Omron Sysmac Studio project TestDataGenerator (Sysmac Studio 1.66.0.7, StandardProject)

# Controller Util: NX102-9000 version 1.64
Task PrimaryTask (priority 4, period or condition 10000): Generate
Library RingBufferLib 0.0.2 (contents left out)
Library FileStreamWriterLib 0.0.2 (contents left out)

TYPE Alignment1Struct : STRUCT  (* Size = 4; Tail Padding = 0; Alignment = 1; Density = 1.000; *)
    aUsint : USINT;  (* Offset = 0; Padding = 0; Size = 1; Alignment = 1; *)
    aSint : SINT;  (* Offset = 1; Padding = 0; Size = 1; Alignment = 1; *)
    Bytes : ARRAY[0..1] OF BYTE;  (* Offset = 2; Padding = 0; Size = 2; Alignment = 1; *)
END_STRUCT END_TYPE
TYPE Alignment2Struct : STRUCT  (* Size = 8; Tail Padding = 0; Alignment = 2; Density = 0.578; *)
    aBool : BOOL;  (* Offset = 0; Padding = 0; Size = 2; Alignment = 2; *)
    aUint : UINT;  (* Offset = 2; Padding = 0; Size = 2; Alignment = 2; *)
    aInt : INT;  (* Offset = 4; Padding = 0; Size = 2; Alignment = 2; *)
    Bools : ARRAY[0..3] OF BOOL;  (* Offset = 6; Padding = 0; Size = 2; Alignment = 2; *)
END_STRUCT END_TYPE
TYPE Alignment4Struct : STRUCT  (* Size = 16; Tail Padding = 0; Alignment = 4; Density = 1.000; *)
    aUdint : UDINT;  (* Offset = 0; Padding = 0; Size = 4; Alignment = 4; *)
    aDint : DINT;  (* Offset = 4; Padding = 0; Size = 4; Alignment = 4; *)
    Uints : ARRAY[0..1] OF UINT;  (* Offset = 8; Padding = 0; Size = 4; Alignment = 2; *)
    Bytes : ARRAY[0..3] OF BYTE;  (* Offset = 12; Padding = 0; Size = 4; Alignment = 1; *)
END_STRUCT END_TYPE
TYPE Alignment8Struct : STRUCT  (* Size = 32; Tail Padding = 0; Alignment = 8; Density = 0.895; *)
    aUlint : ULINT;  (* Offset = 0; Padding = 0; Size = 8; Alignment = 8; *)
    aLint : LINT;  (* Offset = 8; Padding = 0; Size = 8; Alignment = 8; *)
    Udints : ARRAY[0..1] OF UDINT;  (* Offset = 16; Padding = 0; Size = 8; Alignment = 4; *)
    aAlignment2Struct : Alignment2Struct;  (* Offset = 24; Padding = 0; Size = 8; Alignment = 2; *)
END_STRUCT END_TYPE
TYPE SmallStruct : STRUCT  (* Size = 6; Tail Padding = 0; Alignment = 1; Density = 0.857 *)
    u : USINT;  (* Offset = 0; Padding = 0; Size = 1; Alignment = 1; *)
    s : STRING[5];  (* Offset = 1; Padding = 0; Size = 5; Alignment = 1; *)
END_STRUCT END_TYPE
TYPE PaddedStruct : STRUCT  (* Size = 32; Tail Padding = 6; Alignment = 8; Density = 0.466; *)
    aUsint : USINT;  (* Offset = 0; Padding = 0; Size = 1; Alignment = 1; *)
    aUint : UINT;  (* Offset = 2; Padding = 1; Size = 2; Alignment = 2; *)
    aSint : SINT;  (* Offset = 5; Padding = 0; Size = 1; Alignment = 1; *)
    aDint : DINT;  (* Offset = 8; Padding = 2; Size = 4; Alignment = 4; *)
    aUlint : ULINT;  (* Offset = 16; Padding = 4; Size = 8; Alignment = 8; *)
    aBool : BOOL;  (* Offset = 24; Padding = 0; Size = 2; Alignment = 2; *)
END_STRUCT END_TYPE
TYPE UnionStruct : STRUCT  (* Size = 32; Tail Padding = 0; Alignment = 8; Density = 1.000; *)
    Alignment1Unions : ARRAY[0..1] OF Alignment1Union;  (* Offset = 0; Padding = 0; Size = 8; Alignment = 1; *)
    Alignment2Unions : ARRAY[0..1] OF Alignment2Union;  (* Offset = 8; Padding = 0; Size = 8; Alignment = 2; *)
    aAlignment4Union : Alignment4Union;  (* Offset = 16; Padding = 0; Size = 8; Alignment = 4; *)
    aAlignment8Union : Alignment8Union;  (* Offset = 24; Padding = 0; Size = 8; Alignment = 8; *)
END_STRUCT END_TYPE
TYPE ComplexStruct : STRUCT  (* Size = 56; Tail Padding = 4; Alignment = 8; Density = 0.806; *)
    aUsint : USINT;  (* Offset = 0; Padding = 0; Size = 1; Alignment = 1; *)
    Alignment2Structs : ARRAY[0..1] OF Alignment2Struct;  (* Offset = 2; Padding = 1; Size = 16; Alignment = 2; *)
    aAlignment4Union : Alignment4Union;  (* Offset = 20; Padding = 2; Size = 8; Alignment = 4; *)
    aBool : BOOL;  (* Offset = 28; Padding = 0; Size = 2; Alignment = 2; *)
    Lints : ARRAY[0..1] OF LINT;  (* Offset = 32; Padding = 2; Size = 16; Alignment = 8; *)
    aEnum : TestEnum;  (* Offset = 52; Padding = 0; Size = 4; Alignment = 4; *)
END_STRUCT END_TYPE
TYPE Nest1Struct : STRUCT  (* Size = 8; Tail Padding = 0; Alignment = 2; Density = 1.000; *)
    aSmallStruct : SmallStruct;  (* Offset = 0; Padding = 0; Size = 6; Alignment = 1; *)
    aInt : INT;  (* Offset = 6; Padding = 0; Size = 2; Alignment = 2; *)
END_STRUCT END_TYPE
TYPE Nest2Struct : STRUCT  (* Size = 20; Tail Padding = 0; Alignment = 4; Density =0.900; *)
    aNest1Struct : Nest1Struct;  (* Offset = 0; Padding = 0; Size = 8; Alignment = 2; *)
    aSmallStruct : SmallStruct;  (* Offset = 8; Padding = 0; Size = 6; Alignment = 1; *)
    aDint : DINT;  (* Offset = 16; Padding = 2; Size = 4; Alignment = 4; *)
END_STRUCT END_TYPE
TYPE Nest3Struct : STRUCT  (* Size = 40; Tail Padding = 0; Alignment = 8; Density =0.800; *)
    aNest2Struct : Nest2Struct;  (* Offset = 0; Padding = 0; Size = 20; Alignment = 4; *)
    aSmallStruct : SmallStruct;  (* Offset = 20; Padding = 0; Size = 6; Alignment = 1; *)
    aLint : LINT;  (* Offset = 32; Padding = 6; Size = 8; Alignment = 8; *)
END_STRUCT END_TYPE
TYPE ExampleStruct : STRUCT  (* Size = 32; Tail Padding = 4; Alignment = 8; Density =0.875; *)
    Vel : LREAL;  (* Offset = 0; Padding = 0; Size = 8; Alignment = 8; *)
    Trq : LREAL;  (* Offset = 8; Padding = 0; Size = 8; Alignment = 8; *)
    Acc : LREAL;  (* Offset = 16; Padding = 0; Size = 8; Alignment = 8; *)
    StatusCode : DWORD;  (* Offset = 24; Padding = 0; Size = 4; Alignment = 4; *)
END_STRUCT END_TYPE
TYPE Alignment1Union1D : STRUCT
    Unions : ARRAY[0..2] OF Alignment1Union;
END_STRUCT END_TYPE
TYPE Alignment1Union2D : STRUCT
    Unions : ARRAY[0..2,0..2] OF Alignment1Union;
END_STRUCT END_TYPE
TYPE Alignment1Union3D : STRUCT
    Unions : ARRAY[0..2,0..2,0..2] OF Alignment1Union;
END_STRUCT END_TYPE
TYPE Alignment1UnionD1E1 : STRUCT
    Unions : ARRAY[0..0] OF Alignment1Union;
END_STRUCT END_TYPE
TYPE Alignment1UnionD2E1 : STRUCT
    Unions : ARRAY[0..0,0..0] OF Alignment1Union;
END_STRUCT END_TYPE
TYPE Alignment1UnionD3E1 : STRUCT
    Unions : ARRAY[0..0,0..0,0..0] OF Alignment1Union;
END_STRUCT END_TYPE
TYPE Alignment2Union1D : STRUCT
    Unions : ARRAY[0..2] OF Alignment2Union;
END_STRUCT END_TYPE
TYPE Alignment2Union2D : STRUCT
    Unions : ARRAY[0..2,0..2] OF Alignment2Union;
END_STRUCT END_TYPE
TYPE Alignment2Union3D : STRUCT
    Unions : ARRAY[0..2,0..2,0..2] OF Alignment2Union;
END_STRUCT END_TYPE
TYPE Alignment2UnionD1E1 : STRUCT
    Unions : ARRAY[0..0] OF Alignment2Union;
END_STRUCT END_TYPE
TYPE Alignment2UnionD2E1 : STRUCT
    Unions : ARRAY[0..0,0..0] OF Alignment2Union;
END_STRUCT END_TYPE
TYPE Alignment2UnionD3E1 : STRUCT
    Unions : ARRAY[0..0,0..0,0..0] OF Alignment2Union;
END_STRUCT END_TYPE
TYPE Alignment4Union1D : STRUCT
    Unions : ARRAY[0..2] OF Alignment4Union;
END_STRUCT END_TYPE
TYPE Alignment1Union : UNION  (* Size = 4; Padding = 0; Alignment = 1; Density = 1.000 *)
    Bytes : ARRAY[0..3] OF BYTE;  (* Offset = 0; Padding = 0; Size = 4; Alignment = 1; *)
END_UNION END_TYPE
TYPE Alignment2Union : UNION  (* Size = 4; Padding = 0; Alignment = 2; Density = 1.000 *)
    aBool : BOOL;  (* Offset = 0; Padding = 0; Size = 2; Alignment = 2; *)
    Words : ARRAY[0..1] OF WORD;  (* Offset = 0; Padding = 0; Size = 4; Alignment = 2; *)
END_UNION END_TYPE
TYPE Alignment4Union : UNION  (* Size = 8; Padding = 0; Alignment = 4; Density = 1.000 *)
    Bytes : ARRAY[0..3] OF BYTE;  (* Offset = 0; Padding = 0; Size = 4; Alignment = 1; *)
    Dwords : ARRAY[0..1] OF DWORD;  (* Offset = 0; Padding = 0; Size = 8; Alignment = 4; *)
END_UNION END_TYPE
TYPE Alignment8Union : UNION  (* Size = 8; Padding = 0; Alignment = 8; Density = 1.000 *)
    Words : ARRAY[0..3] OF WORD;  (* Offset = 0; Padding = 0; Size = 8; Alignment = 2; *)
    aLword : LWORD;  (* Offset = 0; Padding = 0; Size = 8; Alignment = 8; *)
END_UNION END_TYPE
TYPE MyEnum : (E1 := 0, E2 := 1); END_TYPE
TYPE MyEnum2 : (E2_1 := 0, E2_2 := 1); END_TYPE
TYPE Alignment4Union2D : STRUCT
    Unions : ARRAY[0..2,0..2] OF Alignment4Union;
END_STRUCT END_TYPE
TYPE Alignment4Union3D : STRUCT
    Unions : ARRAY[0..2,0..2,0..2] OF Alignment4Union;
END_STRUCT END_TYPE
TYPE Alignment4UnionD1E1 : STRUCT
    Unions : ARRAY[0..0] OF Alignment4Union;
END_STRUCT END_TYPE
TYPE Alignment4UnionD2E1 : STRUCT
    Unions : ARRAY[0..0,0..0] OF Alignment4Union;
END_STRUCT END_TYPE
TYPE Alignment4UnionD3E1 : STRUCT
    Unions : ARRAY[0..0,0..0,0..0] OF Alignment4Union;
END_STRUCT END_TYPE
TYPE Alignment8Union1D : STRUCT
    Unions : ARRAY[0..2] OF Alignment8Union;
END_STRUCT END_TYPE
TYPE Alignment8Union2D : STRUCT
    Unions : ARRAY[0..2,0..2] OF Alignment8Union;
END_STRUCT END_TYPE
TYPE Alignment8Union3D : STRUCT
    Unions : ARRAY[0..2,0..2,0..2] OF Alignment8Union;
END_STRUCT END_TYPE
TYPE Alignment8UnionD1E1 : STRUCT
    Unions : ARRAY[0..0] OF Alignment8Union;
END_STRUCT END_TYPE
TYPE Alignment8UnionD2E1 : STRUCT
    Unions : ARRAY[0..0,0..0] OF Alignment8Union;
END_STRUCT END_TYPE
TYPE Alignment8UnionD3E1 : STRUCT
    Unions : ARRAY[0..0,0..0,0..0] OF Alignment8Union;
END_STRUCT END_TYPE
TYPE TestEnum : (TE_E0 := 0, TE_E1 := 1); END_TYPE
TYPE ExampleUnion : UNION  (* Size = 4; Padding = 0; Alignment = 4; Density = 1.000 *)
    StatusFlags : ARRAY[0..15] OF BOOL;  (* Offset = 0; Padding = 0; Size = 2; Alignment = 2; *)
    SegmentedStatusCodes : ARRAY[0..1] OF WORD;  (* Offset = 0; Padding = 0; Size = 4; Alignment = 2; *)
    StatusCode : DWORD;  (* Offset = 0; Padding = 0; Size = 4; Alignment = 4; *)
END_UNION END_TYPE

PROGRAM Generate
VAR
    iFileWriteVar : FileWriteVar;
    iFileWriter : stfreakjp\fileio\FileStreamWriter;
END_VAR
VAR CONSTANT
    STATE_INIT : UINT := 0;
    STATE_CREATE_TEST_VAR : UINT := 20;
    STATE_FINALIZE : UINT := 900;
    STATE_DONE : UINT := 1000;
END_VAR
VAR
    WRITE_VAR_BASE_PATH : STRING[65];
    VARS_LIST_PS1 : STRING[65];
    USINT_ARR_D1 : ARRAY[0..2] OF USINT;
    USINT_ARR_D2 : ARRAY[0..2,0..2] OF USINT;
    USINT_ARR_D3 : ARRAY[0..2,0..2,0..2] OF USINT;
    USINT_ARR_D1_E1 : ARRAY[0..0] OF USINT;
    USINT_ARR_D2_E1 : ARRAY[0..0,0..0] OF USINT;
    USINT_ARR_D3_E1 : ARRAY[0..0,0..0,0..0] OF USINT;
    UINT_ARR_D1 : ARRAY[0..2] OF UINT;
    UINT_ARR_D2 : ARRAY[0..2,0..2] OF UINT;
    UINT_ARR_D3 : ARRAY[0..2,0..2,0..2] OF UINT;
    UINT_ARR_D1_E1 : ARRAY[0..0] OF UINT;
    UINT_ARR_D2_E1 : ARRAY[0..0,0..0] OF UINT;
    UINT_ARR_D3_E1 : ARRAY[0..0,0..0,0..0] OF UINT;
    UDINT_ARR_D1 : ARRAY[0..2] OF UDINT;
    UDINT_ARR_D2 : ARRAY[0..2,0..2] OF UDINT;
    UDINT_ARR_D3 : ARRAY[0..2,0..2,0..2] OF UDINT;
    UDINT_ARR_D1_E1 : ARRAY[0..0] OF UDINT;
    UDINT_ARR_D2_E1 : ARRAY[0..0,0..0] OF UDINT;
    UDINT_ARR_D3_E1 : ARRAY[0..0,0..0,0..0] OF UDINT;
    ULINT_ARR_D1 : ARRAY[0..2] OF ULINT;
    ULINT_ARR_D2 : ARRAY[0..2,0..2] OF ULINT;
    ULINT_ARR_D3 : ARRAY[0..2,0..2,0..2] OF ULINT;
    ULINT_ARR_D1_E1 : ARRAY[0..0] OF ULINT;
    ULINT_ARR_D2_E1 : ARRAY[0..0,0..0] OF ULINT;
    ULINT_ARR_D3_E1 : ARRAY[0..0,0..0,0..0] OF ULINT;
    SINT_ARR_D1 : ARRAY[0..2] OF SINT;
    SINT_ARR_D2 : ARRAY[0..2,0..2] OF SINT;
    SINT_ARR_D3 : ARRAY[0..2,0..2,0..2] OF SINT;
    SINT_ARR_D1_E1 : ARRAY[0..0] OF SINT;
    SINT_ARR_D2_E1 : ARRAY[0..0,0..0] OF SINT;
    SINT_ARR_D3_E1 : ARRAY[0..0,0..0,0..0] OF SINT;
    INT_ARR_D1 : ARRAY[0..2] OF INT;
    INT_ARR_D2 : ARRAY[0..2,0..2] OF INT;
    INT_ARR_D3 : ARRAY[0..2,0..2,0..2] OF INT;
    INT_ARR_D1_E1 : ARRAY[0..0] OF INT;
    INT_ARR_D2_E1 : ARRAY[0..0,0..0] OF INT;
    INT_ARR_D3_E1 : ARRAY[0..0,0..0,0..0] OF INT;
    DINT_ARR_D1 : ARRAY[0..2] OF DINT;
    DINT_ARR_D2 : ARRAY[0..2,0..2] OF DINT;
    DINT_ARR_D3 : ARRAY[0..2,0..2,0..2] OF DINT;
    DINT_ARR_D1_E1 : ARRAY[0..0] OF DINT;
    DINT_ARR_D2_E1 : ARRAY[0..0,0..0] OF DINT;
    DINT_ARR_D3_E1 : ARRAY[0..0,0..0,0..0] OF DINT;
    LINT_ARR_D1 : ARRAY[0..2] OF LINT;
    LINT_ARR_D2 : ARRAY[0..2,0..2] OF LINT;
    LINT_ARR_D3 : ARRAY[0..2,0..2,0..2] OF LINT;
    LINT_ARR_D1_E1 : ARRAY[0..0] OF LINT;
    LINT_ARR_D2_E1 : ARRAY[0..0,0..0] OF LINT;
    LINT_ARR_D3_E1 : ARRAY[0..0,0..0,0..0] OF LINT;
    BYTE_ARR_D1 : ARRAY[0..2] OF BYTE;
    BYTE_ARR_D2 : ARRAY[0..2,0..2] OF BYTE;
    BYTE_ARR_D3 : ARRAY[0..2,0..2,0..2] OF BYTE;
    BYTE_ARR_D1_E1 : ARRAY[0..0] OF BYTE;
    BYTE_ARR_D2_E1 : ARRAY[0..0,0..0] OF BYTE;
    BYTE_ARR_D3_E1 : ARRAY[0..0,0..0,0..0] OF BYTE;
    WORD_ARR_D1 : ARRAY[0..2] OF WORD;
    WORD_ARR_D2 : ARRAY[0..2,0..2] OF WORD;
    WORD_ARR_D3 : ARRAY[0..2,0..2,0..2] OF WORD;
    WORD_ARR_D1_E1 : ARRAY[0..0] OF WORD;
    WORD_ARR_D2_E1 : ARRAY[0..0,0..0] OF WORD;
    WORD_ARR_D3_E1 : ARRAY[0..0,0..0,0..0] OF WORD;
    DWORD_ARR_D1 : ARRAY[0..2] OF DWORD;
    DWORD_ARR_D2 : ARRAY[0..2,0..2] OF DWORD;
    DWORD_ARR_D3 : ARRAY[0..2,0..2,0..2] OF DWORD;
    DWORD_ARR_D1_E1 : ARRAY[0..0] OF DWORD;
    DWORD_ARR_D2_E1 : ARRAY[0..0,0..0] OF DWORD;
    DWORD_ARR_D3_E1 : ARRAY[0..0,0..0,0..0] OF DWORD;
    LWORD_ARR_D1 : ARRAY[0..2] OF LWORD;
    LWORD_ARR_D2 : ARRAY[0..2,0..2] OF LWORD;
    LWORD_ARR_D3 : ARRAY[0..2,0..2,0..2] OF LWORD;
    LWORD_ARR_D1_E1 : ARRAY[0..0] OF LWORD;
    LWORD_ARR_D2_E1 : ARRAY[0..0,0..0] OF LWORD;
    LWORD_ARR_D3_E1 : ARRAY[0..0,0..0,0..0] OF LWORD;
    REAL_ARR_D1 : ARRAY[0..2] OF REAL;
    REAL_ARR_D2 : ARRAY[0..2,0..2] OF REAL;
    REAL_ARR_D3 : ARRAY[0..2,0..2,0..2] OF REAL;
    REAL_ARR_D1_E1 : ARRAY[0..0] OF REAL;
    REAL_ARR_D2_E1 : ARRAY[0..0,0..0] OF REAL;
    REAL_ARR_D3_E1 : ARRAY[0..0,0..0,0..0] OF REAL;
    LREAL_ARR_D1 : ARRAY[0..2] OF LREAL;
    LREAL_ARR_D2 : ARRAY[0..2,0..2] OF LREAL;
    LREAL_ARR_D3 : ARRAY[0..2,0..2,0..2] OF LREAL;
    LREAL_ARR_D1_E1 : ARRAY[0..0] OF LREAL;
    LREAL_ARR_D2_E1 : ARRAY[0..0,0..0] OF LREAL;
    LREAL_ARR_D3_E1 : ARRAY[0..0,0..0,0..0] OF LREAL;
    TIME_ARR_D1 : ARRAY[0..2] OF TIME;
    TIME_ARR_D2 : ARRAY[0..2,0..2] OF TIME;
    TIME_ARR_D3 : ARRAY[0..2,0..2,0..2] OF TIME;
    TIME_ARR_D1_E1 : ARRAY[0..0] OF TIME;
    TIME_ARR_D2_E1 : ARRAY[0..0,0..0] OF TIME;
    TIME_ARR_D3_E1 : ARRAY[0..0,0..0,0..0] OF TIME;
    DATE_ARR_D1 : ARRAY[0..2] OF DATE;
    DATE_ARR_D2 : ARRAY[0..2,0..2] OF DATE;
    DATE_ARR_D3 : ARRAY[0..2,0..2,0..2] OF DATE;
    DATE_ARR_D1_E1 : ARRAY[0..0] OF DATE;
    DATE_ARR_D2_E1 : ARRAY[0..0,0..0] OF DATE;
    DATE_ARR_D3_E1 : ARRAY[0..0,0..0,0..0] OF DATE;
    TOD_ARR_D1 : ARRAY[0..2] OF TIME_OF_DAY;
    TOD_ARR_D2 : ARRAY[0..2,0..2] OF TIME_OF_DAY;
    TOD_ARR_D3 : ARRAY[0..2,0..2,0..2] OF TIME_OF_DAY;
    TOD_ARR_D1_E1 : ARRAY[0..0] OF TIME_OF_DAY;
    TOD_ARR_D2_E1 : ARRAY[0..0,0..0] OF TIME_OF_DAY;
    TOD_ARR_D3_E1 : ARRAY[0..0,0..0,0..0] OF TIME_OF_DAY;
    DT_ARR_D1 : ARRAY[0..2] OF DATE_AND_TIME;
    DT_ARR_D2 : ARRAY[0..2,0..2] OF DATE_AND_TIME;
    DT_ARR_D3 : ARRAY[0..2,0..2,0..2] OF DATE_AND_TIME;
    DT_ARR_D1_E1 : ARRAY[0..0] OF DATE_AND_TIME;
    DT_ARR_D2_E1 : ARRAY[0..0,0..0] OF DATE_AND_TIME;
    DT_ARR_D3_E1 : ARRAY[0..0,0..0,0..0] OF DATE_AND_TIME;
    STRING_N2 : STRING[2];
    STRING_N16 : STRING[16];
    BOOL_ARR_D1 : ARRAY[0..2] OF BOOL;
    BOOL_ARR_D2 : ARRAY[0..2,0..2] OF BOOL;
    BOOL_ARR_D3 : ARRAY[0..2,0..2,0..2] OF BOOL;
    BOOL_ARR_D1_E1 : ARRAY[0..0] OF BOOL;
    BOOL_ARR_D2_E1 : ARRAY[0..0,0..0] OF BOOL;
    BOOL_ARR_D3_E1 : ARRAY[0..0,0..0,0..0] OF BOOL;
    STRUCT_ALIGNMENT1 : Alignment1Struct;
    STRUCT_ALIGNMENT1_ARR_D1 : ARRAY[0..2] OF Alignment1Struct;
    STRUCT_ALIGNMENT1_ARR_D1_E1 : ARRAY[0..0] OF Alignment1Struct;
    STRUCT_ALIGNMENT1_ARR_D2_E1 : ARRAY[0..0,0..0] OF Alignment1Struct;
    STRUCT_ALIGNMENT1_ARR_D3_E1 : ARRAY[0..0,0..0,0..0] OF Alignment1Struct;
    STRUCT_ALIGNMENT2 : Alignment2Struct;
    STRUCT_ALIGNMENT2_ARR_D1 : ARRAY[0..2] OF Alignment2Struct;
    STRUCT_ALIGNMENT2_ARR_D1_E1 : ARRAY[0..0] OF Alignment2Struct;
    STRUCT_ALIGNMENT2_ARR_D2_E1 : ARRAY[0..0,0..0] OF Alignment2Struct;
    STRUCT_ALIGNMENT2_ARR_D3_E1 : ARRAY[0..0,0..0,0..0] OF Alignment2Struct;
    STRUCT_ALIGNMENT4 : Alignment4Struct;
    STRUCT_ALIGNMENT8 : Alignment8Struct;
    STRUCT_SMALL : SmallStruct;
    STRUCT_SMALL_ARR_D1 : ARRAY[0..2] OF SmallStruct;
    STRUCT_SMALL_ARR_D2 : ARRAY[0..2,0..2] OF SmallStruct;
    STRUCT_SMALL_ARR_D3 : ARRAY[0..2,0..2,0..2] OF SmallStruct;
    STRUCT_SMALL_ARR_D1_E1 : ARRAY[0..0] OF SmallStruct;
    STRUCT_SMALL_ARR_D2_E1 : ARRAY[0..0,0..0] OF SmallStruct;
    STRUCT_SMALL_ARR_D3_E1 : ARRAY[0..0,0..0,0..0] OF SmallStruct;
    STRUCT_PADDED : PaddedStruct;
    STRUCT_PADDED_ARR_D1 : ARRAY[0..2] OF PaddedStruct;
    STRUCT_PADDED_ARR_D1_E1 : ARRAY[0..0] OF PaddedStruct;
    STRUCT_PADDED_ARR_D2_E1 : ARRAY[0..0,0..0] OF PaddedStruct;
    STRUCT_PADDED_ARR_D3_E1 : ARRAY[0..0,0..0,0..0] OF PaddedStruct;
    UNION_ALIGNMENT1 : Alignment1Union;
    UNION_ALIGNMENT1_ARR_D1 : Alignment1Union1D;
    UNION_ALIGNMENT1_ARR_D2 : ARRAY[0..2,0..2] OF Alignment1Union;
    UNION_ALIGNMENT1_ARR_D3 : ARRAY[0..2,0..2,0..2] OF Alignment1Union;
    UNION_ALIGNMENT2 : Alignment2Union;
    UNION_ALIGNMENT2_ARR_D1 : Alignment2Union1D;
    UNION_ALIGNMENT2_ARR_D2 : Alignment2Union2D;
    UNION_ALIGNMENT2_ARR_D3 : Alignment2Union3D;
    UNION_ALIGNMENT2_ARR_D1_E1 : Alignment2UnionD1E1;
    UNION_ALIGNMENT2_ARR_D2_E1 : Alignment2UnionD2E1;
    UNION_ALIGNMENT2_ARR_D3_E1 : Alignment2UnionD3E1;
    UNION_ALIGNMENT4 : Alignment4Union;
    UNION_ALIGNMENT4_ARR_D1_E1 : Alignment4UnionD1E1;
    UNION_ALIGNMENT4_ARR_D2_E1 : Alignment4UnionD2E1;
    UNION_ALIGNMENT4_ARR_D3_E1 : Alignment4UnionD3E1;
    UNION_ALIGNMENT8 : Alignment8Union;
    UNION_ALIGNMENT8_ARR_D1_E1 : Alignment8UnionD1E1;
    UNION_ALIGNMENT8_ARR_D2_E1 : Alignment8UnionD2E1;
    UNION_ALIGNMENT8_ARR_D3_E1 : Alignment8UnionD3E1;
    STRUCT_UNION : UnionStruct;
    STRUCT_UNION_ARR_D1 : ARRAY[0..2] OF UnionStruct;
    STRUCT_UNION_ARR_D1_E1 : ARRAY[0..0] OF UnionStruct;
    STRUCT_UNION_ARR_D2_E1 : ARRAY[0..0,0..0] OF UnionStruct;
    STRUCT_UNION_ARR_D3_E1 : ARRAY[0..0,0..0,0..0] OF UnionStruct;
    STRUCT_COMPLEX : ComplexStruct;
    STRUCT_NEST2 : Nest2Struct;
    STRUCT_NEST1 : Nest1Struct;
    STRUCT_NEST3 : Nest3Struct;
    STRUCT_EXAMPLE : ExampleStruct;
    UNION_EXAMPLE : ExampleUnion;
    iState : UINT := 0;
    iReturnState : UINT;
    iBufferContext : stfreakjp\buf\RingBufferContext;
    iBuffer : ARRAY[0..65534] OF BYTE;
    iFileWriterContext : stfreakjp\fileio\FileStreamWriterContext;
    iVarIndex : UINT;
    iCurrentVarIndex : UINT;
    iVarName : STRING[256];
    iVarDeclare : STRING[256];
    iVarType : STRING[256];
    iVarAlignmnet : STRING[256];
    iVarCardinalities : STRING[256];
    iVarIsArray : STRING[256];
    iVarKsType : STRING[256];
    iVarKsId : STRING[256];
    iVarKsDefineType : STRING[256];
    iVarKsDefine : STRING[1024];
    iVarBin : ARRAY[0..1023] OF BYTE;
    iVarBinSize : UINT;
    iVarValue : STRING[1986];
    iVarFilePath : STRING[65];
    iTmpStr : STRING[1986];
END_VAR
CASE iState OF
	0:
		iState := STATE_CREATE_TEST_VAR;
		
	// STATE_CREATE_TEST_VAR
	20:
		iFileWriter.Enable := FALSE;

		Clear(iBufferContext);
		Clear(iFileWriterContext);
		
		WRITE_VAR_BASE_PATH := '/testvars/';
		VARS_LIST_PS1 := '/testvars.ps1';
		
		Inc(iState);
	21:
		\\stfreakjp\buf\RingBuffer_init(Context:=iBufferContext,
										Buffer:=iBuffer);
	
		\\stfreakjp\fileio\FileStreamWriter_configure(Context:=iFileWriterContext,
													  Activate:=TRUE,
													  Path:=VARS_LIST_PS1,
													  FileOpenMode:=_eFOPEN_MODE#_WRITE_CREATE,
													  FlushThreshold:=8192,
													  FlushOnDeactivate:=TRUE,
													  RetryTimes:=5,
													  RetryInterval:=5);
		
		iFileWriter.Enable := TRUE;
		
		iVarIndex := 0;
		iCurrentVarIndex := 0;
		
		Inc(iState);
	22:
		iCurrentVarIndex := iVarIndex;
		CASE iVarIndex OF
			// USINT
			0:
				iVarName := 'USINT_ARR_D1_LH';
				iVarDeclare := 'ARRAY[0..2] OF USINT';
				iVarValue := '[0,1,2]';
				iVarKsType := 'nj::usint_array_1d(3)';
				iVarKsId := 'usint_arr_d1_lh';
				
				Clear(USINT_ARR_D1);
				USINT_ARR_D1[0] := 0; USINT_ARR_D1[1] := 1; USINT_ARR_D1[2] := 2;
				iVarBinSize := ToAryByte(In:=USINT_ARR_D1, Order:=_eBYTE_ORDER#_LOW_HIGH, AryOut:=iVarBin[0]);
				Inc(iVarIndex);
			1:
				iVarName := 'USINT_ARR_D2_LH';
				iVarDeclare := 'ARRAY[0..2,0..2] OF USINT';
				iVarValue := '[[0,1,2], [3,4,5], [6,7,8]]';
				iVarKsType := 'nj::usint_array_2d(3,3)';
				iVarKsId := 'usint_arr_d2_lh';
				
				Clear(USINT_ARR_D2);
				USINT_ARR_D2[0, 0] := 0; USINT_ARR_D2[0, 1] := 1; USINT_ARR_D2[0, 2] := 2;
				USINT_ARR_D2[1, 0] := 3; USINT_ARR_D2[1, 1] := 4; USINT_ARR_D2[1, 2] := 5;
				USINT_ARR_D2[2, 0] := 6; USINT_ARR_D2[2, 1] := 7; USINT_ARR_D2[2, 2] := 8;
				iVarBinSize := ToAryByte(In:=USINT_ARR_D2, Order:=_eBYTE_ORDER#_LOW_HIGH, AryOut:=iVarBin[0]);
				Inc(iVarIndex);
			2:
				iVarName := 'USINT_ARR_D3_LH';
				iVarDeclare := 'ARRAY[0..2,0..2,0..2] OF USINT';
				iVarValue := '[[[0,1,2], [3,4,5], [6,7,8]],[[9,10,11], [12,13,14], [15,16,17]],[[18,19,20], [21,22,23], [24,25,26]]]';
				iVarKsType := 'nj::usint_array_3d(3,3,3)';
				iVarKsId := 'usint_arr_d3_lh';
				
				Clear(USINT_ARR_D3);
				USINT_ARR_D3[0, 0, 0] :=  0; USINT_ARR_D3[0, 0, 1] :=  1; USINT_ARR_D3[0, 0, 2] :=  2;
				USINT_ARR_D3[0, 1, 0] :=  3; USINT_ARR_D3[0, 1, 1] :=  4; USINT_ARR_D3[0, 1, 2] :=  5;
				USINT_ARR_D3[0, 2, 0] :=  6; USINT_ARR_D3[0, 2, 1] :=  7; USINT_ARR_D3[0, 2, 2] :=  8;
				USINT_ARR_D3[1, 0, 0] :=  9; USINT_ARR_D3[1, 0, 1] := 10; USINT_ARR_D3[1, 0, 2] := 11;
				USINT_ARR_D3[1, 1, 0] := 12; USINT_ARR_D3[1, 1, 1] := 13; USINT_ARR_D3[1, 1, 2] := 14;
				USINT_ARR_D3[1, 2, 0] := 15; USINT_ARR_D3[1, 2, 1] := 16; USINT_ARR_D3[1, 2, 2] := 17;
				USINT_ARR_D3[2, 0, 0] := 18; USINT_ARR_D3[2, 0, 1] := 19; USINT_ARR_D3[2, 0, 2] := 20;
				USINT_ARR_D3[2, 1, 0] := 21; USINT_ARR_D3[2, 1, 1] := 22; USINT_ARR_D3[2, 1, 2] := 23;
				USINT_ARR_D3[2, 2, 0] := 24; USINT_ARR_D3[2, 2, 1] := 25; USINT_ARR_D3[2, 2, 2] := 26;

				iVarBinSize := ToAryByte(In:=USINT_ARR_D3, Order:=_eBYTE_ORDER#_LOW_HIGH, AryOut:=iVarBin[0]);
				Inc(iVarIndex);
			3:
				iVarName := 'USINT_ARR_D1_E1_LH';
				iVarDeclare := 'ARRAY[0..0] OF USINT';
				iVarValue := '[1]';
				iVarKsType := 'nj::usint_array_1d(1)';
				iVarKsId := 'usint_arr_d1_e1_lh';
				
				Clear(USINT_ARR_D1_E1);
				USINT_ARR_D1_E1[0] := 1;
				iVarBinSize := ToAryByte(In:=USINT_ARR_D1_E1, Order:=_eBYTE_ORDER#_LOW_HIGH, AryOut:=iVarBin[0]);
				Inc(iVarIndex);
			4:
				iVarName := 'USINT_ARR_D2_E1_LH';
				iVarDeclare := 'ARRAY[0..0,0..0] OF USINT';
				iVarValue := '[[1]]';
				iVarKsType := 'nj::usint_array_2d(1,1)';
				iVarKsId := 'usint_arr_d2_e1_lh';
				
				Clear(USINT_ARR_D2_E1);
				USINT_ARR_D2_E1[0, 0] := 1;
				iVarBinSize := ToAryByte(In:=USINT_ARR_D2_E1, Order:=_eBYTE_ORDER#_LOW_HIGH, AryOut:=iVarBin[0]);
				Inc(iVarIndex);
			5:
				iVarName := 'USINT_ARR_D3_E1_LH';
				iVarDeclare := 'ARRAY[0..0,0..0,0..0] OF USINT';
				iVarValue := '[[[1]]]';
				iVarKsType := 'nj::usint_array_3d(1,1,1)';
				iVarKsId := 'usint_arr_d3_e1_lh';
				
				Clear(USINT_ARR_D3_E1);
				USINT_ARR_D3_E1[0, 0, 0] := 1;
				iVarBinSize := ToAryByte(In:=USINT_ARR_D3_E1, Order:=_eBYTE_ORDER#_LOW_HIGH, AryOut:=iVarBin[0]);
				iVarIndex := iVarIndex - iVarIndex MOD 10 + 10;

			// UINT
			10:
				iVarName := 'UINT_ARR_D1_LH';
				iVarDeclare := 'ARRAY[0..2] OF UINT';
				iVarValue := '[0,1,2]';
				iVarKsType := 'nj::uint_array_1d(3)';
				iVarKsId := 'uint_arr_d1_lh';
				
				Clear(UINT_ARR_D1);
				UINT_ARR_D1[0] := 0; UINT_ARR_D1[1] := 1; UINT_ARR_D1[2] := 2;
				iVarBinSize := ToAryByte(In:=UINT_ARR_D1, Order:=_eBYTE_ORDER#_LOW_HIGH, AryOut:=iVarBin[0]);
				Inc(iVarIndex);
			11:
				iVarName := 'UINT_ARR_D2_LH';
				iVarDeclare := 'ARRAY[0..2,0..2] OF UINT';
				iVarValue := '[[0,1,2], [3,4,5], [6,7,8]]';
				iVarKsType := 'nj::uint_array_2d(3,3)';
				iVarKsId := 'uint_arr_d2_lh';
				
				Clear(UINT_ARR_D2);
				UINT_ARR_D2[0, 0] := 0; UINT_ARR_D2[0, 1] := 1; UINT_ARR_D2[0, 2] := 2;
				UINT_ARR_D2[1, 0] := 3; UINT_ARR_D2[1, 1] := 4; UINT_ARR_D2[1, 2] := 5;
				UINT_ARR_D2[2, 0] := 6; UINT_ARR_D2[2, 1] := 7; UINT_ARR_D2[2, 2] := 8;
				iVarBinSize := ToAryByte(In:=UINT_ARR_D2, Order:=_eBYTE_ORDER#_LOW_HIGH, AryOut:=iVarBin[0]);
				Inc(iVarIndex);
			12:
				iVarName := 'UINT_ARR_D3_LH';
				iVarDeclare := 'ARRAY[0..2,0..2,0..2] OF UINT';
				iVarValue := '[[[0,1,2], [3,4,5], [6,7,8]],[[9,10,11], [12,13,14], [15,16,17]],[[18,19,20], [21,22,23], [24,25,26]]]';
				iVarKsType := 'nj::uint_array_3d(3,3,3)';
				iVarKsId := 'uint_arr_d3_lh';
				
				Clear(UINT_ARR_D3);
				UINT_ARR_D3[0, 0, 0] :=  0; UINT_ARR_D3[0, 0, 1] :=  1; UINT_ARR_D3[0, 0, 2] :=  2;
				UINT_ARR_D3[0, 1, 0] :=  3; UINT_ARR_D3[0, 1, 1] :=  4; UINT_ARR_D3[0, 1, 2] :=  5;
				UINT_ARR_D3[0, 2, 0] :=  6; UINT_ARR_D3[0, 2, 1] :=  7; UINT_ARR_D3[0, 2, 2] :=  8;
				UINT_ARR_D3[1, 0, 0] :=  9; UINT_ARR_D3[1, 0, 1] := 10; UINT_ARR_D3[1, 0, 2] := 11;
				UINT_ARR_D3[1, 1, 0] := 12; UINT_ARR_D3[1, 1, 1] := 13; UINT_ARR_D3[1, 1, 2] := 14;
				UINT_ARR_D3[1, 2, 0] := 15; UINT_ARR_D3[1, 2, 1] := 16; UINT_ARR_D3[1, 2, 2] := 17;
				UINT_ARR_D3[2, 0, 0] := 18; UINT_ARR_D3[2, 0, 1] := 19; UINT_ARR_D3[2, 0, 2] := 20;
				UINT_ARR_D3[2, 1, 0] := 21; UINT_ARR_D3[2, 1, 1] := 22; UINT_ARR_D3[2, 1, 2] := 23;
				UINT_ARR_D3[2, 2, 0] := 24; UINT_ARR_D3[2, 2, 1] := 25; UINT_ARR_D3[2, 2, 2] := 26;

				iVarBinSize := ToAryByte(In:=UINT_ARR_D3, Order:=_eBYTE_ORDER#_LOW_HIGH, AryOut:=iVarBin[0]);
				Inc(iVarIndex);
			13:
				iVarName := 'UINT_ARR_D1_E1_LH';
				iVarDeclare := 'ARRAY[0..0] OF UINT';
				iVarValue := '[1]';
				iVarKsType := 'nj::uint_array_1d(1)';
				iVarKsId := 'uint_arr_d1_e1_lh';
				
				Clear(UINT_ARR_D1_E1);
				UINT_ARR_D1_E1[0] := 1;
				iVarBinSize := ToAryByte(In:=UINT_ARR_D1_E1, Order:=_eBYTE_ORDER#_LOW_HIGH, AryOut:=iVarBin[0]);
				Inc(iVarIndex);
			14:
				iVarName := 'UINT_ARR_D2_E1_LH';
				iVarDeclare := 'ARRAY[0..0,0..0] OF UINT';
				iVarValue := '[[1]]';
				iVarKsType := 'nj::uint_array_2d(1,1)';
				iVarKsId := 'uint_arr_d2_e1_lh';
				
				Clear(UINT_ARR_D2_E1);
				UINT_ARR_D2_E1[0, 0] := 1;
				iVarBinSize := ToAryByte(In:=UINT_ARR_D2_E1, Order:=_eBYTE_ORDER#_LOW_HIGH, AryOut:=iVarBin[0]);
				Inc(iVarIndex);
			15:
				iVarName := 'UINT_ARR_D3_E1_LH';
				iVarDeclare := 'ARRAY[0..0,0..0,0..0] OF UINT';
				iVarValue := '[[[1]]]';
				iVarKsType := 'nj::uint_array_3d(1,1,1)';
				iVarKsId := 'uint_arr_d3_lh';
				
				Clear(UINT_ARR_D3_E1);
				UINT_ARR_D3_E1[0, 0, 0] := 1;
				iVarBinSize := ToAryByte(In:=UINT_ARR_D3_E1, Order:=_eBYTE_ORDER#_LOW_HIGH, AryOut:=iVarBin[0]);
				iVarIndex := iVarIndex - iVarIndex MOD 10 + 10;

			// UDINT
			20:
				iVarName := 'UDINT_ARR_D1_LH';
				iVarDeclare := 'ARRAY[0..2] OF UDINT';
				iVarValue := '[0,1,2]';
				iVarKsType := 'nj::udint_array_1d(3)';
				iVarKsId := 'udint_arr_d1_lh';
				
				Clear(UDINT_ARR_D1);
				UDINT_ARR_D1[0] := 0; UDINT_ARR_D1[1] := 1; UDINT_ARR_D1[2] := 2;
				iVarBinSize := ToAryByte(In:=UDINT_ARR_D1, Order:=_eBYTE_ORDER#_LOW_HIGH, AryOut:=iVarBin[0]);
				Inc(iVarIndex);
			21:
				iVarName := 'UDINT_ARR_D2_LH';
				iVarDeclare := 'ARRAY[0..2,0..2] OF UDINT';
				iVarValue := '[[0,1,2], [3,4,5], [6,7,8]]';
				iVarKsType := 'nj::udint_array_2d(3,3)';
				iVarKsId := 'udint_arr_d2_lh';
				
				Clear(UDINT_ARR_D2);
				UDINT_ARR_D2[0, 0] := 0; UDINT_ARR_D2[0, 1] := 1; UDINT_ARR_D2[0, 2] := 2;
				UDINT_ARR_D2[1, 0] := 3; UDINT_ARR_D2[1, 1] := 4; UDINT_ARR_D2[1, 2] := 5;
				UDINT_ARR_D2[2, 0] := 6; UDINT_ARR_D2[2, 1] := 7; UDINT_ARR_D2[2, 2] := 8;
				iVarBinSize := ToAryByte(In:=UDINT_ARR_D2, Order:=_eBYTE_ORDER#_LOW_HIGH, AryOut:=iVarBin[0]);
				Inc(iVarIndex);
			22:
				iVarName := 'UDINT_ARR_D3_LH';
				iVarDeclare := 'ARRAY[0..2,0..2,0..2] OF UDINT';
				iVarValue := '[[[0,1,2], [3,4,5], [6,7,8]],[[9,10,11], [12,13,14], [15,16,17]],[[18,19,20], [21,22,23], [24,25,26]]]';
				iVarKsType := 'nj::udint_array_3d(3,3,3)';
				iVarKsId := 'udint_arr_d3_lh';
				
				Clear(UDINT_ARR_D3);
				UDINT_ARR_D3[0, 0, 0] :=  0; UDINT_ARR_D3[0, 0, 1] :=  1; UDINT_ARR_D3[0, 0, 2] :=  2;
				UDINT_ARR_D3[0, 1, 0] :=  3; UDINT_ARR_D3[0, 1, 1] :=  4; UDINT_ARR_D3[0, 1, 2] :=  5;
				UDINT_ARR_D3[0, 2, 0] :=  6; UDINT_ARR_D3[0, 2, 1] :=  7; UDINT_ARR_D3[0, 2, 2] :=  8;
				UDINT_ARR_D3[1, 0, 0] :=  9; UDINT_ARR_D3[1, 0, 1] := 10; UDINT_ARR_D3[1, 0, 2] := 11;
				UDINT_ARR_D3[1, 1, 0] := 12; UDINT_ARR_D3[1, 1, 1] := 13; UDINT_ARR_D3[1, 1, 2] := 14;
				UDINT_ARR_D3[1, 2, 0] := 15; UDINT_ARR_D3[1, 2, 1] := 16; UDINT_ARR_D3[1, 2, 2] := 17;
				UDINT_ARR_D3[2, 0, 0] := 18; UDINT_ARR_D3[2, 0, 1] := 19; UDINT_ARR_D3[2, 0, 2] := 20;
				UDINT_ARR_D3[2, 1, 0] := 21; UDINT_ARR_D3[2, 1, 1] := 22; UDINT_ARR_D3[2, 1, 2] := 23;
				UDINT_ARR_D3[2, 2, 0] := 24; UDINT_ARR_D3[2, 2, 1] := 25; UDINT_ARR_D3[2, 2, 2] := 26;

				iVarBinSize := ToAryByte(In:=UDINT_ARR_D3, Order:=_eBYTE_ORDER#_LOW_HIGH, AryOut:=iVarBin[0]);
				Inc(iVarIndex);
			23:
				iVarName := 'UDINT_ARR_D1_E1_LH';
				iVarDeclare := 'ARRAY[0..0] OF UDINT';
				iVarValue := '[1]';
				iVarKsType := 'nj::udint_array_1d(1)';
				iVarKsId := 'udint_arr_d1_e1_lh';
				
				Clear(UDINT_ARR_D1_E1);
				UDINT_ARR_D1_E1[0] := 1;
				iVarBinSize := ToAryByte(In:=UDINT_ARR_D1_E1, Order:=_eBYTE_ORDER#_LOW_HIGH, AryOut:=iVarBin[0]);
				Inc(iVarIndex);
			24:
				iVarName := 'UDINT_ARR_D2_E1_LH';
				iVarDeclare := 'ARRAY[0..0,0..0] OF UDINT';
				iVarValue := '[[1]]';
				iVarKsType := 'nj::udint_array_2d(1,1)';
				iVarKsId := 'udint_arr_d2_e1_lh';
				
				Clear(UDINT_ARR_D2_E1);
				UDINT_ARR_D2_E1[0, 0] := 1;
				iVarBinSize := ToAryByte(In:=UDINT_ARR_D2_E1, Order:=_eBYTE_ORDER#_LOW_HIGH, AryOut:=iVarBin[0]);
				Inc(iVarIndex);
			25:
				iVarName := 'UDINT_ARR_D3_E1_LH';
				iVarDeclare := 'ARRAY[0..0,0..0,0..0] OF UDINT';
				iVarValue := '[[[1]]]';
				iVarKsType := 'nj::udint_array_3d(1,1,1)';
				iVarKsId := 'udint_arr_d3_e1_lh';
				
				Clear(UDINT_ARR_D3_E1);
				UDINT_ARR_D3_E1[0, 0, 0] := 1;
				iVarBinSize := ToAryByte(In:=UDINT_ARR_D3_E1, Order:=_eBYTE_ORDER#_LOW_HIGH, AryOut:=iVarBin[0]);
				iVarIndex := iVarIndex - iVarIndex MOD 10 + 10;
				
			// ULINT
			30:
				iVarName := 'ULINT_ARR_D1_LH';
				iVarDeclare := 'ARRAY[0..2] OF ULINT';
				iVarValue := '[0,1,2]';
				iVarKsType := 'nj::ulint_array_1d(3)';
				iVarKsId := 'ulint_arr_d1_lh';
				
				Clear(ULINT_ARR_D1);
				ULINT_ARR_D1[0] := 0; ULINT_ARR_D1[1] := 1; ULINT_ARR_D1[2] := 2;
				iVarBinSize := ToAryByte(In:=ULINT_ARR_D1, Order:=_eBYTE_ORDER#_LOW_HIGH, AryOut:=iVarBin[0]);
				Inc(iVarIndex);
			31:
				iVarName := 'ULINT_ARR_D2_LH';
				iVarDeclare := 'ARRAY[0..2,0..2] OF ULINT';
				iVarValue := '[[0,1,2], [3,4,5], [6,7,8]]';
				iVarKsType := 'nj::ulint_array_2d(3,3)';
				iVarKsId := 'ulint_arr_d2_lh';
				
				Clear(ULINT_ARR_D2);
				ULINT_ARR_D2[0, 0] := 0; ULINT_ARR_D2[0, 1] := 1; ULINT_ARR_D2[0, 2] := 2;
				ULINT_ARR_D2[1, 0] := 3; ULINT_ARR_D2[1, 1] := 4; ULINT_ARR_D2[1, 2] := 5;
				ULINT_ARR_D2[2, 0] := 6; ULINT_ARR_D2[2, 1] := 7; ULINT_ARR_D2[2, 2] := 8;
				iVarBinSize := ToAryByte(In:=ULINT_ARR_D2, Order:=_eBYTE_ORDER#_LOW_HIGH, AryOut:=iVarBin[0]);
				Inc(iVarIndex);
			32:
				iVarName := 'ULINT_ARR_D3_LH';
				iVarDeclare := 'ARRAY[0..2,0..2,0..2] OF ULINT';
				iVarValue := '[[[0,1,2], [3,4,5], [6,7,8]],[[9,10,11], [12,13,14], [15,16,17]],[[18,19,20], [21,22,23], [24,25,26]]]';
				iVarKsType := 'nj::ulint_array_3d(3,3,3)';
				iVarKsId := 'ulint_arr_d3_lh';
				
				Clear(ULINT_ARR_D3);
				ULINT_ARR_D3[0, 0, 0] :=  0; ULINT_ARR_D3[0, 0, 1] :=  1; ULINT_ARR_D3[0, 0, 2] :=  2;
				ULINT_ARR_D3[0, 1, 0] :=  3; ULINT_ARR_D3[0, 1, 1] :=  4; ULINT_ARR_D3[0, 1, 2] :=  5;
				ULINT_ARR_D3[0, 2, 0] :=  6; ULINT_ARR_D3[0, 2, 1] :=  7; ULINT_ARR_D3[0, 2, 2] :=  8;
				ULINT_ARR_D3[1, 0, 0] :=  9; ULINT_ARR_D3[1, 0, 1] := 10; ULINT_ARR_D3[1, 0, 2] := 11;
				ULINT_ARR_D3[1, 1, 0] := 12; ULINT_ARR_D3[1, 1, 1] := 13; ULINT_ARR_D3[1, 1, 2] := 14;
				ULINT_ARR_D3[1, 2, 0] := 15; ULINT_ARR_D3[1, 2, 1] := 16; ULINT_ARR_D3[1, 2, 2] := 17;
				ULINT_ARR_D3[2, 0, 0] := 18; ULINT_ARR_D3[2, 0, 1] := 19; ULINT_ARR_D3[2, 0, 2] := 20;
				ULINT_ARR_D3[2, 1, 0] := 21; ULINT_ARR_D3[2, 1, 1] := 22; ULINT_ARR_D3[2, 1, 2] := 23;
				ULINT_ARR_D3[2, 2, 0] := 24; ULINT_ARR_D3[2, 2, 1] := 25; ULINT_ARR_D3[2, 2, 2] := 26;
				iVarBinSize := ToAryByte(In:=ULINT_ARR_D3, Order:=_eBYTE_ORDER#_LOW_HIGH, AryOut:=iVarBin[0]);
				Inc(iVarIndex);
			33:
				iVarName := 'ULINT_ARR_D1_E1_LH';
				iVarDeclare := 'ARRAY[0..0] OF ULINT';
				iVarValue := '[1]';
				iVarKsType := 'nj::ulint_array_1d(1)';
				iVarKsId := 'ulint_arr_d1_e1_lh';
				
				Clear(ULINT_ARR_D1_E1);
				ULINT_ARR_D1_E1[0] := 1;
				iVarBinSize := ToAryByte(In:=ULINT_ARR_D1_E1, Order:=_eBYTE_ORDER#_LOW_HIGH, AryOut:=iVarBin[0]);
				Inc(iVarIndex);
			34:
				iVarName := 'ULINT_ARR_D2_E1_LH';
				iVarDeclare := 'ARRAY[0..0,0..0] OF ULINT';
				iVarValue := '[[1]]';
				iVarKsType := 'nj::ulint_array_2d(1,1)';
				iVarKsId := 'ulint_arr_d2_e1_lh';
				
				Clear(ULINT_ARR_D2_E1);
				ULINT_ARR_D2_E1[0, 0] := 1;
				iVarBinSize := ToAryByte(In:=ULINT_ARR_D2_E1, Order:=_eBYTE_ORDER#_LOW_HIGH, AryOut:=iVarBin[0]);
				Inc(iVarIndex);
			35:
				iVarName := 'ULINT_ARR_D3_E1_LH';
				iVarDeclare := 'ARRAY[0..0,0..0,0..0] OF ULINT';
				iVarValue := '[[[1]]]';
				iVarKsType := 'nj::ulint_array_3d(1,1,1)';
				iVarKsId := 'ulint_arr_d3_e1_lh';
				
				Clear(ULINT_ARR_D3_E1);
				ULINT_ARR_D3_E1[0, 0, 0] := 1;
				iVarBinSize := ToAryByte(In:=ULINT_ARR_D3_E1, Order:=_eBYTE_ORDER#_LOW_HIGH, AryOut:=iVarBin[0]);
				iVarIndex := iVarIndex - iVarIndex MOD 10 + 10;

			// SINT
			40:
				iVarName := 'SINT_ARR_D1_LH';
				iVarDeclare := 'ARRAY[0..2] OF SINT';
				iVarValue := '[0,-1,2]';
				iVarKsType := 'nj::sint_array_1d(3)';
				iVarKsId := 'sint_arr_d1_lh';
				
				Clear(SINT_ARR_D1);
				SINT_ARR_D1[0] := 0; SINT_ARR_D1[1] := -1; SINT_ARR_D1[2] := 2;
				iVarBinSize := ToAryByte(In:=SINT_ARR_D1, Order:=_eBYTE_ORDER#_LOW_HIGH, AryOut:=iVarBin[0]);
				Inc(iVarIndex);
			41:
				iVarName := 'SINT_ARR_D2_LH';
				iVarDeclare := 'ARRAY[0..2,0..2] OF SINT';
				iVarValue := '[[0,-1,2], [-3,4,-5], [6,-7,8]]';
				iVarKsType := 'nj::sint_array_2d(3,3)';
				iVarKsId := 'sint_arr_d2_lh';
				
				Clear(SINT_ARR_D2);
				SINT_ARR_D2[0, 0] := 0; SINT_ARR_D2[0, 1] := -1; SINT_ARR_D2[0, 2] := 2;
				SINT_ARR_D2[1, 0] := -3; SINT_ARR_D2[1, 1] := 4; SINT_ARR_D2[1, 2] := -5;
				SINT_ARR_D2[2, 0] := 6; SINT_ARR_D2[2, 1] := -7; SINT_ARR_D2[2, 2] := 8;
				iVarBinSize := ToAryByte(In:=SINT_ARR_D2, Order:=_eBYTE_ORDER#_LOW_HIGH, AryOut:=iVarBin[0]);
				Inc(iVarIndex);
			42:
				iVarName := 'SINT_ARR_D3_LH';
				iVarDeclare := 'ARRAY[0..2,0..2,0..2] OF SINT';
				iVarValue := '[[[0,-1,2], [-3,4,-5], [6,-7,8]],[[-9,10,-11], [12,-13,14], [-15,16,-17]],[[18,-19,20], [-21,22,-23], [24,-25,26]]]';
				iVarKsType := 'nj::sint_array_3d(3,3,3)';
				iVarKsId := 'sint_arr_d3_lh';
				
				Clear(SINT_ARR_D3);
				SINT_ARR_D3[0, 0, 0] :=   0; SINT_ARR_D3[0, 0, 1] :=  -1; SINT_ARR_D3[0, 0, 2] :=   2;
				SINT_ARR_D3[0, 1, 0] :=  -3; SINT_ARR_D3[0, 1, 1] :=   4; SINT_ARR_D3[0, 1, 2] :=  -5;
				SINT_ARR_D3[0, 2, 0] :=   6; SINT_ARR_D3[0, 2, 1] :=  -7; SINT_ARR_D3[0, 2, 2] :=   8;
				SINT_ARR_D3[1, 0, 0] :=  -9; SINT_ARR_D3[1, 0, 1] :=  10; SINT_ARR_D3[1, 0, 2] := -11;
				SINT_ARR_D3[1, 1, 0] :=  12; SINT_ARR_D3[1, 1, 1] := -13; SINT_ARR_D3[1, 1, 2] :=  14;
				SINT_ARR_D3[1, 2, 0] := -15; SINT_ARR_D3[1, 2, 1] :=  16; SINT_ARR_D3[1, 2, 2] := -17;
				SINT_ARR_D3[2, 0, 0] :=  18; SINT_ARR_D3[2, 0, 1] := -19; SINT_ARR_D3[2, 0, 2] :=  20;
				SINT_ARR_D3[2, 1, 0] := -21; SINT_ARR_D3[2, 1, 1] :=  22; SINT_ARR_D3[2, 1, 2] := -23;
				SINT_ARR_D3[2, 2, 0] :=  24; SINT_ARR_D3[2, 2, 1] := -25; SINT_ARR_D3[2, 2, 2] :=  26;
				iVarBinSize := ToAryByte(In:=SINT_ARR_D3, Order:=_eBYTE_ORDER#_LOW_HIGH, AryOut:=iVarBin[0]);
				Inc(iVarIndex);
			43:
				iVarName := 'SINT_ARR_D1_E1_LH';
				iVarDeclare := 'ARRAY[0..0] OF SINT';
				iVarValue := '[-1]';
				iVarKsType := 'nj::sint_array_1d(1)';
				iVarKsId := 'sint_arr_d1_e1_lh';
				
				Clear(SINT_ARR_D1_E1);
				SINT_ARR_D1_E1[0] := -1;
				iVarBinSize := ToAryByte(In:=SINT_ARR_D1_E1, Order:=_eBYTE_ORDER#_LOW_HIGH, AryOut:=iVarBin[0]);
				Inc(iVarIndex);
			44:
				iVarName := 'SINT_ARR_D2_E1_LH';
				iVarDeclare := 'ARRAY[0..0,0..0] OF SINT';
				iVarValue := '[[-1]]';
				iVarKsType := 'nj::sint_array_2d(1,1)';
				iVarKsId := 'sint_arr_d2_e1_lh';
				
				Clear(SINT_ARR_D2_E1);
				SINT_ARR_D2_E1[0, 0] := -1;
				iVarBinSize := ToAryByte(In:=SINT_ARR_D2_E1, Order:=_eBYTE_ORDER#_LOW_HIGH, AryOut:=iVarBin[0]);
				Inc(iVarIndex);
			45:
				iVarName := 'SINT_ARR_D3_E1_LH';
				iVarDeclare := 'ARRAY[0..0,0..0,0..0] OF SINT';
				iVarValue := '[[[-1]]]';
				iVarKsType := 'nj::sint_array_3d(1,1,1)';
				iVarKsId := 'sint_arr_d3_e1_lh';
				
				Clear(SINT_ARR_D3_E1);
				SINT_ARR_D3_E1[0, 0, 0] := -1;
				iVarBinSize := ToAryByte(In:=SINT_ARR_D3_E1, Order:=_eBYTE_ORDER#_LOW_HIGH, AryOut:=iVarBin[0]);
				iVarIndex := iVarIndex - iVarIndex MOD 10 + 10;

			// INT
			50:
				iVarName := 'INT_ARR_D1_LH';
				iVarDeclare := 'ARRAY[0..2] OF INT';
				iVarValue := '[0,-1,2]';
				iVarKsType := 'nj::int_array_1d(3)';
				iVarKsId := 'int_arr_d1_lh';
				
				Clear(INT_ARR_D1);
				INT_ARR_D1[0] := 0; INT_ARR_D1[1] := -1; INT_ARR_D1[2] := 2;
				iVarBinSize := ToAryByte(In:=INT_ARR_D1, Order:=_eBYTE_ORDER#_LOW_HIGH, AryOut:=iVarBin[0]);
				Inc(iVarIndex);
			51:
				iVarName := 'INT_ARR_D2_LH';
				iVarDeclare := 'ARRAY[0..2,0..2] OF INT';
				iVarValue := '[[0,-1,2], [-3,4,-5], [6,-7,8]]';
				iVarKsType := 'nj::int_array_2d(3,3)';
				iVarKsId := 'int_arr_d2_lh';
				
				Clear(INT_ARR_D2);
				INT_ARR_D2[0, 0] := 0; INT_ARR_D2[0, 1] := -1; INT_ARR_D2[0, 2] := 2;
				INT_ARR_D2[1, 0] := -3; INT_ARR_D2[1, 1] := 4; INT_ARR_D2[1, 2] := -5;
				INT_ARR_D2[2, 0] := 6; INT_ARR_D2[2, 1] := -7; INT_ARR_D2[2, 2] := 8;
				iVarBinSize := ToAryByte(In:=INT_ARR_D2, Order:=_eBYTE_ORDER#_LOW_HIGH, AryOut:=iVarBin[0]);
				Inc(iVarIndex);
			52:
				iVarName := 'INT_ARR_D3_LH';
				iVarDeclare := 'ARRAY[0..2,0..2,0..2] OF INT';
				iVarValue := '[[[0,-1,2], [-3,4,-5], [6,-7,8]],[[-9,10,-11], [12,-13,14], [-15,16,-17]],[[18,-19,20], [-21,22,-23], [24,-25,26]]]';
				iVarKsType := 'nj::int_array_3d(3,3,3)';
				iVarKsId := 'int_arr_d3_lh';
				
				Clear(INT_ARR_D3);
				INT_ARR_D3[0, 0, 0] :=   0; INT_ARR_D3[0, 0, 1] :=  -1; INT_ARR_D3[0, 0, 2] :=   2;
				INT_ARR_D3[0, 1, 0] :=  -3; INT_ARR_D3[0, 1, 1] :=   4; INT_ARR_D3[0, 1, 2] :=  -5;
				INT_ARR_D3[0, 2, 0] :=   6; INT_ARR_D3[0, 2, 1] :=  -7; INT_ARR_D3[0, 2, 2] :=   8;
				INT_ARR_D3[1, 0, 0] :=  -9; INT_ARR_D3[1, 0, 1] :=  10; INT_ARR_D3[1, 0, 2] := -11;
				INT_ARR_D3[1, 1, 0] :=  12; INT_ARR_D3[1, 1, 1] := -13; INT_ARR_D3[1, 1, 2] :=  14;
				INT_ARR_D3[1, 2, 0] := -15; INT_ARR_D3[1, 2, 1] :=  16; INT_ARR_D3[1, 2, 2] := -17;
				INT_ARR_D3[2, 0, 0] :=  18; INT_ARR_D3[2, 0, 1] := -19; INT_ARR_D3[2, 0, 2] :=  20;
				INT_ARR_D3[2, 1, 0] := -21; INT_ARR_D3[2, 1, 1] :=  22; INT_ARR_D3[2, 1, 2] := -23;
				INT_ARR_D3[2, 2, 0] :=  24; INT_ARR_D3[2, 2, 1] := -25; INT_ARR_D3[2, 2, 2] :=  26;
				iVarBinSize := ToAryByte(In:=INT_ARR_D3, Order:=_eBYTE_ORDER#_LOW_HIGH, AryOut:=iVarBin[0]);
				Inc(iVarIndex);
			53:
				iVarName := 'INT_ARR_D1_E1_LH';
				iVarDeclare := 'ARRAY[0..0] OF INT';
				iVarValue := '[-1]';
				iVarKsType := 'nj::int_array_1d(1)';
				iVarKsId := 'int_arr_d1_e1_lh';
				
				Clear(INT_ARR_D1_E1);
				INT_ARR_D1_E1[0] := -1;
				iVarBinSize := ToAryByte(In:=INT_ARR_D1_E1, Order:=_eBYTE_ORDER#_LOW_HIGH, AryOut:=iVarBin[0]);
				Inc(iVarIndex);
			54:
				iVarName := 'INT_ARR_D2_E1_LH';
				iVarDeclare := 'ARRAY[0..0,0..0] OF INT';
				iVarValue := '[[-1]]';
				iVarKsType := 'nj::int_array_2d(1,1)';
				iVarKsId := 'int_arr_d2_e1_lh';
				
				Clear(INT_ARR_D2_E1);
				INT_ARR_D2_E1[0, 0] := -1;
				iVarBinSize := ToAryByte(In:=INT_ARR_D2_E1, Order:=_eBYTE_ORDER#_LOW_HIGH, AryOut:=iVarBin[0]);
				Inc(iVarIndex);
			55:
				iVarName := 'INT_ARR_D3_E1_LH';
				iVarDeclare := 'ARRAY[0..0,0..0,0..0] OF INT';
				iVarValue := '[[[-1]]]';
				iVarKsType := 'nj::int_array_3d(1,1,1)';
				iVarKsId := 'int_arr_d3_e1_lh';
				
				Clear(INT_ARR_D3_E1);
				INT_ARR_D3_E1[0, 0, 0] := -1;
				iVarBinSize := ToAryByte(In:=INT_ARR_D3_E1, Order:=_eBYTE_ORDER#_LOW_HIGH, AryOut:=iVarBin[0]);
				iVarIndex := iVarIndex - iVarIndex MOD 10 + 10;
				
			// DINT
			60:
				iVarName := 'DINT_ARR_D1_LH';
				iVarDeclare := 'ARRAY[0..2] OF DINT';
				iVarValue := '[0,-1,2]';
				iVarKsType := 'nj::dint_array_1d(3)';
				iVarKsId := 'dint_arr_d1_lh';
				
				Clear(DINT_ARR_D1);
				DINT_ARR_D1[0] := 0; DINT_ARR_D1[1] := -1; DINT_ARR_D1[2] := 2;
				iVarBinSize := ToAryByte(In:=DINT_ARR_D1, Order:=_eBYTE_ORDER#_LOW_HIGH, AryOut:=iVarBin[0]);
				Inc(iVarIndex);
			61:
				iVarName := 'DINT_ARR_D2_LH';
				iVarDeclare := 'ARRAY[0..2,0..2] OF DINT';
				iVarValue := '[[0,-1,2], [-3,4,-5], [6,-7,8]]';
				iVarKsType := 'nj::dint_array_2d(3,3)';
				iVarKsId := 'dint_arr_d2_lh';
				
				Clear(DINT_ARR_D2);
				DINT_ARR_D2[0, 0] := 0; DINT_ARR_D2[0, 1] := -1; DINT_ARR_D2[0, 2] := 2;
				DINT_ARR_D2[1, 0] := -3; DINT_ARR_D2[1, 1] := 4; DINT_ARR_D2[1, 2] := -5;
				DINT_ARR_D2[2, 0] := 6; DINT_ARR_D2[2, 1] := -7; DINT_ARR_D2[2, 2] := 8;
				iVarBinSize := ToAryByte(In:=DINT_ARR_D2, Order:=_eBYTE_ORDER#_LOW_HIGH, AryOut:=iVarBin[0]);
				Inc(iVarIndex);
			62:
				iVarName := 'DINT_ARR_D3_LH';
				iVarDeclare := 'ARRAY[0..2,0..2,0..2] OF DINT';
				iVarValue := '[[[0,-1,2], [-3,4,-5], [6,-7,8]],[[-9,10,-11], [12,-13,14], [-15,16,-17]],[[18,-19,20], [-21,22,-23], [24,-25,26]]]';
				iVarKsType := 'nj::dint_array_3d(3,3,3)';
				iVarKsId := 'dint_arr_d3_lh';
				
				Clear(DINT_ARR_D3);
				DINT_ARR_D3[0, 0, 0] :=   0; DINT_ARR_D3[0, 0, 1] :=  -1; DINT_ARR_D3[0, 0, 2] :=   2;
				DINT_ARR_D3[0, 1, 0] :=  -3; DINT_ARR_D3[0, 1, 1] :=   4; DINT_ARR_D3[0, 1, 2] :=  -5;
				DINT_ARR_D3[0, 2, 0] :=   6; DINT_ARR_D3[0, 2, 1] :=  -7; DINT_ARR_D3[0, 2, 2] :=   8;
				DINT_ARR_D3[1, 0, 0] :=  -9; DINT_ARR_D3[1, 0, 1] :=  10; DINT_ARR_D3[1, 0, 2] := -11;
				DINT_ARR_D3[1, 1, 0] :=  12; DINT_ARR_D3[1, 1, 1] := -13; DINT_ARR_D3[1, 1, 2] :=  14;
				DINT_ARR_D3[1, 2, 0] := -15; DINT_ARR_D3[1, 2, 1] :=  16; DINT_ARR_D3[1, 2, 2] := -17;
				DINT_ARR_D3[2, 0, 0] :=  18; DINT_ARR_D3[2, 0, 1] := -19; DINT_ARR_D3[2, 0, 2] :=  20;
				DINT_ARR_D3[2, 1, 0] := -21; DINT_ARR_D3[2, 1, 1] :=  22; DINT_ARR_D3[2, 1, 2] := -23;
				DINT_ARR_D3[2, 2, 0] :=  24; DINT_ARR_D3[2, 2, 1] := -25; DINT_ARR_D3[2, 2, 2] :=  26;
				iVarBinSize := ToAryByte(In:=DINT_ARR_D3, Order:=_eBYTE_ORDER#_LOW_HIGH, AryOut:=iVarBin[0]);
				Inc(iVarIndex);
			63:
				iVarName := 'DINT_ARR_D1_E1_LH';
				iVarDeclare := 'ARRAY[0..0] OF DINT';
				iVarValue := '[-1]';
				iVarKsType := 'nj::dint_array_1d(1)';
				iVarKsId := 'dint_arr_d1_e1_lh';
				
				Clear(DINT_ARR_D1_E1);
				DINT_ARR_D1_E1[0] := -1;
				iVarBinSize := ToAryByte(In:=DINT_ARR_D1_E1, Order:=_eBYTE_ORDER#_LOW_HIGH, AryOut:=iVarBin[0]);
				Inc(iVarIndex);
			64:
				iVarName := 'DINT_ARR_D2_E1_LH';
				iVarDeclare := 'ARRAY[0..0,0..0] OF DINT';
				iVarValue := '[[-1]]';
				iVarKsType := 'nj::dint_array_2d(1,1)';
				iVarKsId := 'dint_arr_d2_e1_lh';
				
				Clear(DINT_ARR_D2_E1);
				DINT_ARR_D2_E1[0, 0] := -1;
				iVarBinSize := ToAryByte(In:=DINT_ARR_D2_E1, Order:=_eBYTE_ORDER#_LOW_HIGH, AryOut:=iVarBin[0]);
				Inc(iVarIndex);
			65:
				iVarName := 'DINT_ARR_D3_E1_LH';
				iVarDeclare := 'ARRAY[0..0,0..0,0..0] OF DINT';
				iVarValue := '[[[-1]]]';
				iVarKsType := 'nj::dint_array_3d(1,1,1)';
				iVarKsId := 'dint_arr_d3_e1_lh';
				
				Clear(DINT_ARR_D3_E1);
				DINT_ARR_D3_E1[0, 0, 0] := -1;
				iVarBinSize := ToAryByte(In:=DINT_ARR_D3_E1, Order:=_eBYTE_ORDER#_LOW_HIGH, AryOut:=iVarBin[0]);
				iVarIndex := iVarIndex - iVarIndex MOD 10 + 10;

			// LINT
			70:
				iVarName := 'LINT_ARR_D1_LH';
				iVarDeclare := 'ARRAY[0..2] OF LINT';
				iVarValue := '[0,-1,2]';
				iVarKsType := 'nj::lint_array_1d(3)';
				iVarKsId := 'lint_arr_d1_lh';
				
				Clear(LINT_ARR_D1);
				LINT_ARR_D1[0] := 0; LINT_ARR_D1[1] := -1; LINT_ARR_D1[2] := 2;
				iVarBinSize := ToAryByte(In:=LINT_ARR_D1, Order:=_eBYTE_ORDER#_LOW_HIGH, AryOut:=iVarBin[0]);
				Inc(iVarIndex);
			71:
				iVarName := 'LINT_ARR_D2_LH';
				iVarDeclare := 'ARRAY[0..2,0..2] OF LINT';
				iVarValue := '[[0,-1,2], [-3,4,-5], [6,-7,8]]';
				iVarKsType := 'nj::lint_array_2d(3,3)';
				iVarKsId := 'lint_arr_d2_lh';
				
				Clear(LINT_ARR_D2);
				LINT_ARR_D2[0, 0] := 0; LINT_ARR_D2[0, 1] := -1; LINT_ARR_D2[0, 2] := 2;
				LINT_ARR_D2[1, 0] := -3; LINT_ARR_D2[1, 1] := 4; LINT_ARR_D2[1, 2] := -5;
				LINT_ARR_D2[2, 0] := 6; LINT_ARR_D2[2, 1] := -7; LINT_ARR_D2[2, 2] := 8;
				iVarBinSize := ToAryByte(In:=LINT_ARR_D2, Order:=_eBYTE_ORDER#_LOW_HIGH, AryOut:=iVarBin[0]);
				Inc(iVarIndex);
			72:
				iVarName := 'LINT_ARR_D3_LH';
				iVarDeclare := 'ARRAY[0..2,0..2,0..2] OF LINT';
				iVarValue := '[[[0,-1,2], [-3,4,-5], [6,-7,8]],[[-9,10,-11], [12,-13,14], [-15,16,-17]],[[18,-19,20], [-21,22,-23], [24,-25,26]]]';
				iVarKsType := 'nj::lint_array_3d(3,3,3)';
				iVarKsId := 'lint_arr_d3_lh';
				
				Clear(LINT_ARR_D3);
				LINT_ARR_D3[0, 0, 0] :=   0; LINT_ARR_D3[0, 0, 1] :=  -1; LINT_ARR_D3[0, 0, 2] :=   2;
				LINT_ARR_D3[0, 1, 0] :=  -3; LINT_ARR_D3[0, 1, 1] :=   4; LINT_ARR_D3[0, 1, 2] :=  -5;
				LINT_ARR_D3[0, 2, 0] :=   6; LINT_ARR_D3[0, 2, 1] :=  -7; LINT_ARR_D3[0, 2, 2] :=   8;
				LINT_ARR_D3[1, 0, 0] :=  -9; LINT_ARR_D3[1, 0, 1] :=  10; LINT_ARR_D3[1, 0, 2] := -11;
				LINT_ARR_D3[1, 1, 0] :=  12; LINT_ARR_D3[1, 1, 1] := -13; LINT_ARR_D3[1, 1, 2] :=  14;
				LINT_ARR_D3[1, 2, 0] := -15; LINT_ARR_D3[1, 2, 1] :=  16; LINT_ARR_D3[1, 2, 2] := -17;
				LINT_ARR_D3[2, 0, 0] :=  18; LINT_ARR_D3[2, 0, 1] := -19; LINT_ARR_D3[2, 0, 2] :=  20;
				LINT_ARR_D3[2, 1, 0] := -21; LINT_ARR_D3[2, 1, 1] :=  22; LINT_ARR_D3[2, 1, 2] := -23;
				LINT_ARR_D3[2, 2, 0] :=  24; LINT_ARR_D3[2, 2, 1] := -25; LINT_ARR_D3[2, 2, 2] :=  26;
				iVarBinSize := ToAryByte(In:=LINT_ARR_D3, Order:=_eBYTE_ORDER#_LOW_HIGH, AryOut:=iVarBin[0]);
				Inc(iVarIndex);
			73:
				iVarName := 'LINT_ARR_D1_E1_LH';
				iVarDeclare := 'ARRAY[0..0] OF LINT';
				iVarValue := '[-1]';
				iVarKsType := 'nj::lint_array_1d(1)';
				iVarKsId := 'lint_arr_d1_e1_lh';
				
				Clear(LINT_ARR_D1_E1);
				LINT_ARR_D1_E1[0] := -1;
				iVarBinSize := ToAryByte(In:=LINT_ARR_D1_E1, Order:=_eBYTE_ORDER#_LOW_HIGH, AryOut:=iVarBin[0]);
				Inc(iVarIndex);
			74:
				iVarName := 'LINT_ARR_D2_E1_LH';
				iVarDeclare := 'ARRAY[0..0,0..0] OF LINT';
				iVarValue := '[[-1]]';
				iVarKsType := 'nj::lint_array_2d(1,1)';
				iVarKsId := 'lint_arr_d2_e1_lh';
				
				Clear(LINT_ARR_D2_E1);
				LINT_ARR_D2_E1[0, 0] := -1;
				iVarBinSize := ToAryByte(In:=LINT_ARR_D2_E1, Order:=_eBYTE_ORDER#_LOW_HIGH, AryOut:=iVarBin[0]);
				Inc(iVarIndex);
			75:
				iVarName := 'LINT_ARR_D3_E1_LH';
				iVarDeclare := 'ARRAY[0..0,0..0,0..0] OF LINT';
				iVarValue := '[[[-1]]]';
				iVarKsType := 'nj::lint_array_3d(1,1,1)';
				iVarKsId := 'lint_arr_d3_e1_lh';
				
				Clear(LINT_ARR_D3_E1);
				LINT_ARR_D3_E1[0, 0, 0] := -1;
				iVarBinSize := ToAryByte(In:=LINT_ARR_D3_E1, Order:=_eBYTE_ORDER#_LOW_HIGH, AryOut:=iVarBin[0]);
				iVarIndex := iVarIndex - iVarIndex MOD 10 + 10;
				
			// BYTE
			80:
				iVarName := 'BYTE_ARR_D1_LH';
				iVarDeclare := 'ARRAY[0..2] OF BYTE';
				iVarValue := '[0,1,2]';
				iVarKsType := 'nj::byte_array_1d(3)';
				iVarKsId := 'byte_arr_d1_lh';
				
				Clear(BYTE_ARR_D1);
				BYTE_ARR_D1[0] := 0; BYTE_ARR_D1[1] := 1; BYTE_ARR_D1[2] := 2;
				iVarBinSize := ToAryByte(In:=BYTE_ARR_D1, Order:=_eBYTE_ORDER#_LOW_HIGH, AryOut:=iVarBin[0]);
				Inc(iVarIndex);
			81:
				iVarName := 'BYTE_ARR_D2_LH';
				iVarDeclare := 'ARRAY[0..2,0..2] OF BYTE';
				iVarValue := '[[0,1,2], [3,4,5], [6,7,8]]';
				iVarKsType := 'nj::byte_array_2d(3,3)';
				iVarKsId := 'byte_arr_d2_lh';
				
				Clear(BYTE_ARR_D2);
				BYTE_ARR_D2[0, 0] := 0; BYTE_ARR_D2[0, 1] := 1; BYTE_ARR_D2[0, 2] := 2;
				BYTE_ARR_D2[1, 0] := 3; BYTE_ARR_D2[1, 1] := 4; BYTE_ARR_D2[1, 2] := 5;
				BYTE_ARR_D2[2, 0] := 6; BYTE_ARR_D2[2, 1] := 7; BYTE_ARR_D2[2, 2] := 8;
				iVarBinSize := ToAryByte(In:=BYTE_ARR_D2, Order:=_eBYTE_ORDER#_LOW_HIGH, AryOut:=iVarBin[0]);
				Inc(iVarIndex);
			82:
				iVarName := 'BYTE_ARR_D3_LH';
				iVarDeclare := 'ARRAY[0..2,0..2,0..2] OF BYTE';
				iVarValue := '[[[0,1,2], [3,4,5], [6,7,8]],[[9,10,11], [12,13,14], [15,16,17]],[[18,19,20], [21,22,23], [24,25,26]]]';
				iVarKsType := 'nj::byte_array_3d(3,3,3)';
				iVarKsId := 'byte_arr_d3_lh';
				
				Clear(BYTE_ARR_D3);
				BYTE_ARR_D3[0, 0, 0] :=  0; BYTE_ARR_D3[0, 0, 1] :=  1; BYTE_ARR_D3[0, 0, 2] :=  2;
				BYTE_ARR_D3[0, 1, 0] :=  3; BYTE_ARR_D3[0, 1, 1] :=  4; BYTE_ARR_D3[0, 1, 2] :=  5;
				BYTE_ARR_D3[0, 2, 0] :=  6; BYTE_ARR_D3[0, 2, 1] :=  7; BYTE_ARR_D3[0, 2, 2] :=  8;
				BYTE_ARR_D3[1, 0, 0] :=  9; BYTE_ARR_D3[1, 0, 1] := 10; BYTE_ARR_D3[1, 0, 2] := 11;
				BYTE_ARR_D3[1, 1, 0] := 12; BYTE_ARR_D3[1, 1, 1] := 13; BYTE_ARR_D3[1, 1, 2] := 14;
				BYTE_ARR_D3[1, 2, 0] := 15; BYTE_ARR_D3[1, 2, 1] := 16; BYTE_ARR_D3[1, 2, 2] := 17;
				BYTE_ARR_D3[2, 0, 0] := 18; BYTE_ARR_D3[2, 0, 1] := 19; BYTE_ARR_D3[2, 0, 2] := 20;
				BYTE_ARR_D3[2, 1, 0] := 21; BYTE_ARR_D3[2, 1, 1] := 22; BYTE_ARR_D3[2, 1, 2] := 23;
				BYTE_ARR_D3[2, 2, 0] := 24; BYTE_ARR_D3[2, 2, 1] := 25; BYTE_ARR_D3[2, 2, 2] := 26;

				iVarBinSize := ToAryByte(In:=BYTE_ARR_D3, Order:=_eBYTE_ORDER#_LOW_HIGH, AryOut:=iVarBin[0]);
				Inc(iVarIndex);
			83:
				iVarName := 'BYTE_ARR_D1_E1_LH';
				iVarDeclare := 'ARRAY[0..0] OF BYTE';
				iVarValue := '[1]';
				iVarKsType := 'nj::byte_array_1d(1)';
				iVarKsId := 'byte_arr_d1_e1_lh';
				
				Clear(BYTE_ARR_D1_E1);
				BYTE_ARR_D1_E1[0] := 1;
				iVarBinSize := ToAryByte(In:=BYTE_ARR_D1_E1, Order:=_eBYTE_ORDER#_LOW_HIGH, AryOut:=iVarBin[0]);
				Inc(iVarIndex);
			84:
				iVarName := 'BYTE_ARR_D2_E1_LH';
				iVarDeclare := 'ARRAY[0..0,0..0] OF BYTE';
				iVarValue := '[[1]]';
				iVarKsType := 'nj::byte_array_2d(1,1)';
				iVarKsId := 'byte_arr_d2_e1_lh';
				
				Clear(BYTE_ARR_D2_E1);
				BYTE_ARR_D2_E1[0, 0] := 1;
				iVarBinSize := ToAryByte(In:=BYTE_ARR_D2_E1, Order:=_eBYTE_ORDER#_LOW_HIGH, AryOut:=iVarBin[0]);
				Inc(iVarIndex);
			85:
				iVarName := 'BYTE_ARR_D3_E1_LH';
				iVarDeclare := 'ARRAY[0..0,0..0,0..0] OF BYTE';
				iVarValue := '[[[1]]]';
				iVarKsType := 'nj::byte_array_3d(1,1,1)';
				iVarKsId := 'byte_arr_d3_e1_lh';
				
				Clear(BYTE_ARR_D3_E1);
				BYTE_ARR_D3_E1[0, 0, 0] := 1;
				iVarBinSize := ToAryByte(In:=BYTE_ARR_D3_E1, Order:=_eBYTE_ORDER#_LOW_HIGH, AryOut:=iVarBin[0]);
				iVarIndex := iVarIndex - iVarIndex MOD 10 + 10;

			// WORD
			90:
				iVarName := 'WORD_ARR_D1_LH';
				iVarDeclare := 'ARRAY[0..2] OF WORD';
				iVarValue := '[0,1,2]';
				iVarKsType := 'nj::word_array_1d(3)';
				iVarKsId := 'word_arr_d1_lh';
				
				Clear(WORD_ARR_D1);
				WORD_ARR_D1[0] := 0; WORD_ARR_D1[1] := 1; WORD_ARR_D1[2] := 2;
				iVarBinSize := ToAryByte(In:=WORD_ARR_D1, Order:=_eBYTE_ORDER#_LOW_HIGH, AryOut:=iVarBin[0]);
				Inc(iVarIndex);
			91:
				iVarName := 'WORD_ARR_D2_LH';
				iVarDeclare := 'ARRAY[0..2,0..2] OF WORD';
				iVarValue := '[[0,1,2], [3,4,5], [6,7,8]]';
				iVarKsType := 'nj::word_array_2d(3,3)';
				iVarKsId := 'word_arr_d2_lh';
				
				Clear(WORD_ARR_D2);
				WORD_ARR_D2[0, 0] := 0; WORD_ARR_D2[0, 1] := 1; WORD_ARR_D2[0, 2] := 2;
				WORD_ARR_D2[1, 0] := 3; WORD_ARR_D2[1, 1] := 4; WORD_ARR_D2[1, 2] := 5;
				WORD_ARR_D2[2, 0] := 6; WORD_ARR_D2[2, 1] := 7; WORD_ARR_D2[2, 2] := 8;
				iVarBinSize := ToAryByte(In:=WORD_ARR_D2, Order:=_eBYTE_ORDER#_LOW_HIGH, AryOut:=iVarBin[0]);
				Inc(iVarIndex);
			92:
				iVarName := 'WORD_ARR_D3_LH';
				iVarDeclare := 'ARRAY[0..2,0..2,0..2] OF WORD';
				iVarValue := '[[[0,1,2], [3,4,5], [6,7,8]],[[9,10,11], [12,13,14], [15,16,17]],[[18,19,20], [21,22,23], [24,25,26]]]';
				iVarKsType := 'nj::word_array_3d(3,3,3)';
				iVarKsId := 'word_arr_d3_lh';
				
				Clear(WORD_ARR_D3);
				WORD_ARR_D3[0, 0, 0] :=  0; WORD_ARR_D3[0, 0, 1] :=  1; WORD_ARR_D3[0, 0, 2] :=  2;
				WORD_ARR_D3[0, 1, 0] :=  3; WORD_ARR_D3[0, 1, 1] :=  4; WORD_ARR_D3[0, 1, 2] :=  5;
				WORD_ARR_D3[0, 2, 0] :=  6; WORD_ARR_D3[0, 2, 1] :=  7; WORD_ARR_D3[0, 2, 2] :=  8;
				WORD_ARR_D3[1, 0, 0] :=  9; WORD_ARR_D3[1, 0, 1] := 10; WORD_ARR_D3[1, 0, 2] := 11;
				WORD_ARR_D3[1, 1, 0] := 12; WORD_ARR_D3[1, 1, 1] := 13; WORD_ARR_D3[1, 1, 2] := 14;
				WORD_ARR_D3[1, 2, 0] := 15; WORD_ARR_D3[1, 2, 1] := 16; WORD_ARR_D3[1, 2, 2] := 17;
				WORD_ARR_D3[2, 0, 0] := 18; WORD_ARR_D3[2, 0, 1] := 19; WORD_ARR_D3[2, 0, 2] := 20;
				WORD_ARR_D3[2, 1, 0] := 21; WORD_ARR_D3[2, 1, 1] := 22; WORD_ARR_D3[2, 1, 2] := 23;
				WORD_ARR_D3[2, 2, 0] := 24; WORD_ARR_D3[2, 2, 1] := 25; WORD_ARR_D3[2, 2, 2] := 26;

				iVarBinSize := ToAryByte(In:=WORD_ARR_D3, Order:=_eBYTE_ORDER#_LOW_HIGH, AryOut:=iVarBin[0]);
				Inc(iVarIndex);
			93:
				iVarName := 'WORD_ARR_D1_E1_LH';
				iVarDeclare := 'ARRAY[0..0] OF WORD';
				iVarValue := '[1]';
				iVarKsType := 'nj::word_array_1d(1)';
				iVarKsId := 'word_arr_d1_e1_lh';
				
				Clear(WORD_ARR_D1_E1);
				WORD_ARR_D1_E1[0] := 1;
				iVarBinSize := ToAryByte(In:=WORD_ARR_D1_E1, Order:=_eBYTE_ORDER#_LOW_HIGH, AryOut:=iVarBin[0]);
				Inc(iVarIndex);
			94:
				iVarName := 'WORD_ARR_D2_E1_LH';
				iVarDeclare := 'ARRAY[0..0,0..0] OF WORD';
				iVarValue := '[[1]]';
				iVarKsType := 'nj::word_array_2d(1,1)';
				iVarKsId := 'word_arr_d2_e1_lh';
				
				Clear(WORD_ARR_D2_E1);
				WORD_ARR_D2_E1[0, 0] := 1;
				iVarBinSize := ToAryByte(In:=WORD_ARR_D2_E1, Order:=_eBYTE_ORDER#_LOW_HIGH, AryOut:=iVarBin[0]);
				Inc(iVarIndex);
			95:
				iVarName := 'WORD_ARR_D3_E1_LH';
				iVarDeclare := 'ARRAY[0..0,0..0,0..0] OF WORD';
				iVarValue := '[[[1]]]';
				iVarKsType := 'nj::word_array_3d(1,1,1)';
				iVarKsId := 'word_arr_d3_e1_lh';
				
				Clear(WORD_ARR_D3_E1);
				WORD_ARR_D3_E1[0, 0, 0] := 1;
				iVarBinSize := ToAryByte(In:=WORD_ARR_D3_E1, Order:=_eBYTE_ORDER#_LOW_HIGH, AryOut:=iVarBin[0]);
				iVarIndex := iVarIndex - iVarIndex MOD 10 + 10;

			// DWORD:
			100:
				iVarName := 'DWORD_ARR_D1_LH';
				iVarDeclare := 'ARRAY[0..2] OF DWORD';
				iVarValue := '[0,1,2]';
				iVarKsType := 'nj::dword_array_1d(3)';
				iVarKsId := 'dword_arr_d1_lh';
				
				Clear(DWORD_ARR_D1);
				DWORD_ARR_D1[0] := 0; DWORD_ARR_D1[1] := 1; DWORD_ARR_D1[2] := 2;
				iVarBinSize := ToAryByte(In:=DWORD_ARR_D1, Order:=_eBYTE_ORDER#_LOW_HIGH, AryOut:=iVarBin[0]);
				Inc(iVarIndex);
			101:
				iVarName := 'DWORD_ARR_D2_LH';
				iVarDeclare := 'ARRAY[0..2,0..2] OF DWORD';
				iVarValue := '[[0,1,2], [3,4,5], [6,7,8]]';
				iVarKsType := 'nj::dword_array_2d(3,3)';
				iVarKsId := 'dword_arr_d2_lh';
				
				Clear(DWORD_ARR_D2);
				DWORD_ARR_D2[0, 0] := 0; DWORD_ARR_D2[0, 1] := 1; DWORD_ARR_D2[0, 2] := 2;
				DWORD_ARR_D2[1, 0] := 3; DWORD_ARR_D2[1, 1] := 4; DWORD_ARR_D2[1, 2] := 5;
				DWORD_ARR_D2[2, 0] := 6; DWORD_ARR_D2[2, 1] := 7; DWORD_ARR_D2[2, 2] := 8;
				iVarBinSize := ToAryByte(In:=DWORD_ARR_D2, Order:=_eBYTE_ORDER#_LOW_HIGH, AryOut:=iVarBin[0]);
				Inc(iVarIndex);
			102:
				iVarName := 'DWORD_ARR_D3_LH';
				iVarDeclare := 'ARRAY[0..2,0..2,0..2] OF DWORD';
				iVarValue := '[[[0,1,2], [3,4,5], [6,7,8]],[[9,10,11], [12,13,14], [15,16,17]],[[18,19,20], [21,22,23], [24,25,26]]]';
				iVarKsType := 'nj::dword_array_3d(3,3,3)';
				iVarKsId := 'dword_arr_d3_lh';
				
				Clear(DWORD_ARR_D3);
				DWORD_ARR_D3[0, 0, 0] :=  0; DWORD_ARR_D3[0, 0, 1] :=  1; DWORD_ARR_D3[0, 0, 2] :=  2;
				DWORD_ARR_D3[0, 1, 0] :=  3; DWORD_ARR_D3[0, 1, 1] :=  4; DWORD_ARR_D3[0, 1, 2] :=  5;
				DWORD_ARR_D3[0, 2, 0] :=  6; DWORD_ARR_D3[0, 2, 1] :=  7; DWORD_ARR_D3[0, 2, 2] :=  8;
				DWORD_ARR_D3[1, 0, 0] :=  9; DWORD_ARR_D3[1, 0, 1] := 10; DWORD_ARR_D3[1, 0, 2] := 11;
				DWORD_ARR_D3[1, 1, 0] := 12; DWORD_ARR_D3[1, 1, 1] := 13; DWORD_ARR_D3[1, 1, 2] := 14;
				DWORD_ARR_D3[1, 2, 0] := 15; DWORD_ARR_D3[1, 2, 1] := 16; DWORD_ARR_D3[1, 2, 2] := 17;
				DWORD_ARR_D3[2, 0, 0] := 18; DWORD_ARR_D3[2, 0, 1] := 19; DWORD_ARR_D3[2, 0, 2] := 20;
				DWORD_ARR_D3[2, 1, 0] := 21; DWORD_ARR_D3[2, 1, 1] := 22; DWORD_ARR_D3[2, 1, 2] := 23;
				DWORD_ARR_D3[2, 2, 0] := 24; DWORD_ARR_D3[2, 2, 1] := 25; DWORD_ARR_D3[2, 2, 2] := 26;

				iVarBinSize := ToAryByte(In:=DWORD_ARR_D3, Order:=_eBYTE_ORDER#_LOW_HIGH, AryOut:=iVarBin[0]);
				Inc(iVarIndex);
			103:
				iVarName := 'DWORD_ARR_D1_E1_LH';
				iVarDeclare := 'ARRAY[0..0] OF DWORD';
				iVarValue := '[1]';
				iVarKsType := 'nj::dword_array_1d(1)';
				iVarKsId := 'dword_arr_d1_e1_lh';
				
				Clear(DWORD_ARR_D1_E1);
				DWORD_ARR_D1_E1[0] := 1;
				iVarBinSize := ToAryByte(In:=DWORD_ARR_D1_E1, Order:=_eBYTE_ORDER#_LOW_HIGH, AryOut:=iVarBin[0]);
				Inc(iVarIndex);
			104:
				iVarName := 'DWORD_ARR_D2_E1_LH';
				iVarDeclare := 'ARRAY[0..0,0..0] OF DWORD';
				iVarValue := '[[1]]';
				iVarKsType := 'nj::dword_array_2d(1,1)';
				iVarKsId := 'dword_arr_d2_e1_lh';
				
				Clear(DWORD_ARR_D2_E1);
				DWORD_ARR_D2_E1[0, 0] := 1;
				iVarBinSize := ToAryByte(In:=DWORD_ARR_D2_E1, Order:=_eBYTE_ORDER#_LOW_HIGH, AryOut:=iVarBin[0]);
				Inc(iVarIndex);
			105:
				iVarName := 'DWORD_ARR_D3_E1_LH';
				iVarDeclare := 'ARRAY[0..0,0..0,0..0] OF DWORD';
				iVarValue := '[[[1]]]';
				iVarKsType := 'nj::dword_array_3d(1,1,1)';
				iVarKsId := 'dword_arr_d3_e1_lh';
				
				Clear(DWORD_ARR_D3_E1);
				DWORD_ARR_D3_E1[0, 0, 0] := 1;
				iVarBinSize := ToAryByte(In:=DWORD_ARR_D3_E1, Order:=_eBYTE_ORDER#_LOW_HIGH, AryOut:=iVarBin[0]);
				iVarIndex := iVarIndex - iVarIndex MOD 10 + 10;
				
			// LWORD:
			110:
				iVarName := 'LWORD_ARR_D1_LH';
				iVarDeclare := 'ARRAY[0..2] OF LWORD';
				iVarValue := '[0,1,2]';
				iVarKsType := 'nj::lword_array_1d(3)';
				iVarKsId := 'lword_arr_d1_lh';
				
				Clear(LWORD_ARR_D1);
				LWORD_ARR_D1[0] := 0; LWORD_ARR_D1[1] := 1; LWORD_ARR_D1[2] := 2;
				iVarBinSize := ToAryByte(In:=LWORD_ARR_D1, Order:=_eBYTE_ORDER#_LOW_HIGH, AryOut:=iVarBin[0]);
				Inc(iVarIndex);
			111:
				iVarName := 'LWORD_ARR_D2_LH';
				iVarDeclare := 'ARRAY[0..2,0..2] OF LWORD';
				iVarValue := '[[0,1,2], [3,4,5], [6,7,8]]';
				iVarKsType := 'nj::lword_array_2d(3,3)';
				iVarKsId := 'lword_arr_d2_lh';
				
				Clear(LWORD_ARR_D2);
				LWORD_ARR_D2[0, 0] := 0; LWORD_ARR_D2[0, 1] := 1; LWORD_ARR_D2[0, 2] := 2;
				LWORD_ARR_D2[1, 0] := 3; LWORD_ARR_D2[1, 1] := 4; LWORD_ARR_D2[1, 2] := 5;
				LWORD_ARR_D2[2, 0] := 6; LWORD_ARR_D2[2, 1] := 7; LWORD_ARR_D2[2, 2] := 8;
				iVarBinSize := ToAryByte(In:=LWORD_ARR_D2, Order:=_eBYTE_ORDER#_LOW_HIGH, AryOut:=iVarBin[0]);
				Inc(iVarIndex);
			112:
				iVarName := 'LWORD_ARR_D3_LH';
				iVarDeclare := 'ARRAY[0..2,0..2,0..2] OF LWORD';
				iVarValue := '[[[0,1,2], [3,4,5], [6,7,8]],[[9,10,11], [12,13,14], [15,16,17]],[[18,19,20], [21,22,23], [24,25,26]]]';
				iVarKsType := 'nj::lword_array_3d(3,3,3)';
				iVarKsId := 'lword_arr_d3_lh';
				
				Clear(LWORD_ARR_D3);
				LWORD_ARR_D3[0, 0, 0] :=  0; LWORD_ARR_D3[0, 0, 1] :=  1; LWORD_ARR_D3[0, 0, 2] :=  2;
				LWORD_ARR_D3[0, 1, 0] :=  3; LWORD_ARR_D3[0, 1, 1] :=  4; LWORD_ARR_D3[0, 1, 2] :=  5;
				LWORD_ARR_D3[0, 2, 0] :=  6; LWORD_ARR_D3[0, 2, 1] :=  7; LWORD_ARR_D3[0, 2, 2] :=  8;
				LWORD_ARR_D3[1, 0, 0] :=  9; LWORD_ARR_D3[1, 0, 1] := 10; LWORD_ARR_D3[1, 0, 2] := 11;
				LWORD_ARR_D3[1, 1, 0] := 12; LWORD_ARR_D3[1, 1, 1] := 13; LWORD_ARR_D3[1, 1, 2] := 14;
				LWORD_ARR_D3[1, 2, 0] := 15; LWORD_ARR_D3[1, 2, 1] := 16; LWORD_ARR_D3[1, 2, 2] := 17;
				LWORD_ARR_D3[2, 0, 0] := 18; LWORD_ARR_D3[2, 0, 1] := 19; LWORD_ARR_D3[2, 0, 2] := 20;
				LWORD_ARR_D3[2, 1, 0] := 21; LWORD_ARR_D3[2, 1, 1] := 22; LWORD_ARR_D3[2, 1, 2] := 23;
				LWORD_ARR_D3[2, 2, 0] := 24; LWORD_ARR_D3[2, 2, 1] := 25; LWORD_ARR_D3[2, 2, 2] := 26;
				iVarBinSize := ToAryByte(In:=LWORD_ARR_D3, Order:=_eBYTE_ORDER#_LOW_HIGH, AryOut:=iVarBin[0]);
				Inc(iVarIndex);
			113:
				iVarName := 'LWORD_ARR_D1_E1_LH';
				iVarDeclare := 'ARRAY[0..0] OF LWORD';
				iVarValue := '[1]';
				iVarKsType := 'nj::lword_array_1d(1)';
				iVarKsId := 'lword_arr_d1_e1_lh';
				
				Clear(LWORD_ARR_D1_E1);
				LWORD_ARR_D1_E1[0] := 1;
				iVarBinSize := ToAryByte(In:=LWORD_ARR_D1_E1, Order:=_eBYTE_ORDER#_LOW_HIGH, AryOut:=iVarBin[0]);
				Inc(iVarIndex);
			114:
				iVarName := 'LWORD_ARR_D2_E1_LH';
				iVarDeclare := 'ARRAY[0..0,0..0] OF LWORD';
				iVarValue := '[[1]]';
				iVarKsType := 'nj::lword_array_2d(1,1)';
				iVarKsId := 'lword_arr_d2_e1_lh';
				
				Clear(LWORD_ARR_D2_E1);
				LWORD_ARR_D2_E1[0, 0] := 1;
				iVarBinSize := ToAryByte(In:=LWORD_ARR_D2_E1, Order:=_eBYTE_ORDER#_LOW_HIGH, AryOut:=iVarBin[0]);
				Inc(iVarIndex);
			115:
				iVarName := 'LWORD_ARR_D3_E1_LH';
				iVarDeclare := 'ARRAY[0..0,0..0,0..0] OF LWORD';
				iVarValue := '[[[1]]]';
				iVarKsType := 'nj::lword_array_3d(1,1,1)';
				iVarKsId := 'lword_arr_d3_e1_lh';
				
				Clear(LWORD_ARR_D3_E1);
				LWORD_ARR_D3_E1[0, 0, 0] := 1;
				iVarBinSize := ToAryByte(In:=LWORD_ARR_D3_E1, Order:=_eBYTE_ORDER#_LOW_HIGH, AryOut:=iVarBin[0]);
				iVarIndex := iVarIndex - iVarIndex MOD 10 + 10;

			// REAL
			120:
				iVarName := 'REAL_ARR_D1_LH';
				iVarDeclare := 'ARRAY[0..2] OF REAL';
				iVarValue := '[0,1.0,2.0]';
				iVarKsType := 'nj::real_array_1d(3)';
				iVarKsId := 'real_arr_d1_lh';
				
				Clear(REAL_ARR_D1);
				REAL_ARR_D1[0] := 0; REAL_ARR_D1[1] := 1.0; REAL_ARR_D1[2] := 2.0;
				iVarBinSize := ToAryByte(In:=REAL_ARR_D1, Order:=_eBYTE_ORDER#_LOW_HIGH, AryOut:=iVarBin[0]);
				Inc(iVarIndex);
			121:
				iVarName := 'REAL_ARR_D2_LH';
				iVarDeclare := 'ARRAY[0..2,0..2] OF REAL';
				iVarValue := '[[0,1.0,2.0], [4.0,8.0,16.0], [32.0,64.0,128.0]]';
				iVarKsType := 'nj::real_array_2d(3,3)';
				iVarKsId := 'real_arr_d2_lh';
				
				Clear(REAL_ARR_D2);
				REAL_ARR_D2[0, 0] := 0; REAL_ARR_D2[0, 1] := 1; REAL_ARR_D2[0, 2] := 2;
				REAL_ARR_D2[1, 0] := 4; REAL_ARR_D2[1, 1] := 8; REAL_ARR_D2[1, 2] := 16;
				REAL_ARR_D2[2, 0] := 32; REAL_ARR_D2[2, 1] := 64; REAL_ARR_D2[2, 2] := 128;
				iVarBinSize := ToAryByte(In:=REAL_ARR_D2, Order:=_eBYTE_ORDER#_LOW_HIGH, AryOut:=iVarBin[0]);
				Inc(iVarIndex);
			122:
				iVarName := 'REAL_ARR_D3_LH';
				iVarDeclare := 'ARRAY[0..2,0..2,0..2] OF REAL';
				iVarValue := '[[[0,1.0,2.0], [4.0,8.0,16.0], [32.0,64.0,128.0]],[[256.0,512.0,1024.0], [2048.0,0.5,0.25],[0.125,0.0625,0.03125]],[[0.015625,0.0078125,0.00390625],[0.001953125,0.0009765625,0.00048828125],[0.000244140625,-1.0,-0.5]]]';
				iVarKsType := 'nj::real_array_3d(3,3,3)';
				iVarKsId := 'real_arr_d3_lh';
				
				Clear(REAL_ARR_D3);
				REAL_ARR_D3[0, 0, 0] :=  0; REAL_ARR_D3[0, 0, 1] :=  1.0; REAL_ARR_D3[0, 0, 2] :=  2.0;
				REAL_ARR_D3[0, 1, 0] :=  4.0; REAL_ARR_D3[0, 1, 1] :=  8.0; REAL_ARR_D3[0, 1, 2] :=  16.0;
				REAL_ARR_D3[0, 2, 0] :=  32.0; REAL_ARR_D3[0, 2, 1] :=  64.0; REAL_ARR_D3[0, 2, 2] :=  128.0;
				REAL_ARR_D3[1, 0, 0] :=  256.0; REAL_ARR_D3[1, 0, 1] := 512.0; REAL_ARR_D3[1, 0, 2] := 1024.0;
				REAL_ARR_D3[1, 1, 0] := 2048.0; REAL_ARR_D3[1, 1, 1] := 0.5; REAL_ARR_D3[1, 1, 2] := 0.25;
				REAL_ARR_D3[1, 2, 0] := 0.125; REAL_ARR_D3[1, 2, 1] := 0.0625; REAL_ARR_D3[1, 2, 2] := 0.03125;
				REAL_ARR_D3[2, 0, 0] := 0.015625; REAL_ARR_D3[2, 0, 1] := 0.0078125; REAL_ARR_D3[2, 0, 2] := 0.00390625;
				REAL_ARR_D3[2, 1, 0] := 0.001953125; REAL_ARR_D3[2, 1, 1] := 0.0009765625; REAL_ARR_D3[2, 1, 2] := 0.00048828125;
				REAL_ARR_D3[2, 2, 0] := 0.000244140625; REAL_ARR_D3[2, 2, 1] := -1.0; REAL_ARR_D3[2, 2, 2] := -0.5;
				iVarBinSize := ToAryByte(In:=REAL_ARR_D3, Order:=_eBYTE_ORDER#_LOW_HIGH, AryOut:=iVarBin[0]);
				Inc(iVarIndex);
			123:
				iVarName := 'REAL_ARR_D1_E1_LH';
				iVarDeclare := 'ARRAY[0..0] OF REAL';
				iVarValue := '[1.0]';
				iVarKsType := 'nj::real_array_1d(1)';
				iVarKsId := 'real_arr_d1_e1_lh';
				
				Clear(REAL_ARR_D1_E1);
				REAL_ARR_D1_E1[0] := 1.0;
				iVarBinSize := ToAryByte(In:=REAL_ARR_D1_E1, Order:=_eBYTE_ORDER#_LOW_HIGH, AryOut:=iVarBin[0]);
				Inc(iVarIndex);
			124:
				iVarName := 'REAL_ARR_D2_E1_LH';
				iVarDeclare := 'ARRAY[0..0,0..0] OF REAL';
				iVarValue := '[[1.0]]';
				iVarKsType := 'nj::real_array_2d(1,1)';
				iVarKsId := 'real_arr_d2_e1_lh';
				
				Clear(REAL_ARR_D2_E1);
				REAL_ARR_D2_E1[0, 0] := 1.0;
				iVarBinSize := ToAryByte(In:=REAL_ARR_D2_E1, Order:=_eBYTE_ORDER#_LOW_HIGH, AryOut:=iVarBin[0]);
				Inc(iVarIndex);
			125:
				iVarName := 'REAL_ARR_D3_E1_LH';
				iVarDeclare := 'ARRAY[0..0,0..0,0..0] OF REAL';
				iVarValue := '[[[1.0]]]';
				iVarKsType := 'nj::real_array_3d(1,1,1)';
				iVarKsId := 'real_arr_d3_e1_lh';
				
				Clear(REAL_ARR_D3_E1);
				REAL_ARR_D3_E1[0, 0, 0] := 1.0;
				iVarBinSize := ToAryByte(In:=REAL_ARR_D3_E1, Order:=_eBYTE_ORDER#_LOW_HIGH, AryOut:=iVarBin[0]);
				iVarIndex := iVarIndex - iVarIndex MOD 10 + 10;

			// LREAL
			130:
				iVarName := 'LREAL_ARR_D1_LH';
				iVarDeclare := 'ARRAY[0..2] OF LREAL';
				iVarValue := '[0,1.0,2.0]';
				iVarKsType := 'nj::lreal_array_1d(3)';
				iVarKsId := 'lreal_arr_d1_lh';
				
				Clear(LREAL_ARR_D1);
				LREAL_ARR_D1[0] := 0; LREAL_ARR_D1[1] := 1.0; LREAL_ARR_D1[2] := 2.0;
				iVarBinSize := ToAryByte(In:=LREAL_ARR_D1, Order:=_eBYTE_ORDER#_LOW_HIGH, AryOut:=iVarBin[0]);
				Inc(iVarIndex);
			131:
				iVarName := 'LREAL_ARR_D2_LH';
				iVarDeclare := 'ARRAY[0..2,0..2] OF LREAL';
				iVarValue := '[[0,1.0,2.0], [4.0,8.0,16.0], [32.0,64.0,128.0]]';
				iVarKsType := 'nj::lreal_array_2d(3,3)';
				iVarKsId := 'lreal_arr_d2_lh';
				
				Clear(LREAL_ARR_D2);
				LREAL_ARR_D2[0, 0] := 0; LREAL_ARR_D2[0, 1] := 1; LREAL_ARR_D2[0, 2] := 2;
				LREAL_ARR_D2[1, 0] := 4; LREAL_ARR_D2[1, 1] := 8; LREAL_ARR_D2[1, 2] := 16;
				LREAL_ARR_D2[2, 0] := 32; LREAL_ARR_D2[2, 1] := 64; LREAL_ARR_D2[2, 2] := 128;
				iVarBinSize := ToAryByte(In:=LREAL_ARR_D2, Order:=_eBYTE_ORDER#_LOW_HIGH, AryOut:=iVarBin[0]);
				Inc(iVarIndex);
			132:
				iVarName := 'LREAL_ARR_D3_LH';
				iVarDeclare := 'ARRAY[0..2,0..2,0..2] OF LREAL';
				iVarValue := '[[[0,1.0,2.0], [4.0,8.0,16.0], [32.0,64.0,128.0]],[[256.0,512.0,1024.0], [2048.0,0.5,0.25],[0.125,0.0625,0.03125]],[[0.015625,0.0078125,0.00390625],[0.001953125,0.0009765625,0.00048828125],[0.000244140625,-1.0,-0.5]]]';
				iVarKsType := 'nj::lreal_array_3d(3,3,3)';
				iVarKsId := 'lreal_arr_d3_lh';
				
				Clear(LREAL_ARR_D3);
				LREAL_ARR_D3[0, 0, 0] :=  0; LREAL_ARR_D3[0, 0, 1] :=  1.0; LREAL_ARR_D3[0, 0, 2] :=  2.0;
				LREAL_ARR_D3[0, 1, 0] :=  4.0; LREAL_ARR_D3[0, 1, 1] :=  8.0; LREAL_ARR_D3[0, 1, 2] :=  16.0;
				LREAL_ARR_D3[0, 2, 0] :=  32.0; LREAL_ARR_D3[0, 2, 1] :=  64.0; LREAL_ARR_D3[0, 2, 2] :=  128.0;
				LREAL_ARR_D3[1, 0, 0] :=  256.0; LREAL_ARR_D3[1, 0, 1] := 512.0; LREAL_ARR_D3[1, 0, 2] := 1024.0;
				LREAL_ARR_D3[1, 1, 0] := 2048.0; LREAL_ARR_D3[1, 1, 1] := 0.5; LREAL_ARR_D3[1, 1, 2] := 0.25;
				LREAL_ARR_D3[1, 2, 0] := 0.125; LREAL_ARR_D3[1, 2, 1] := 0.0625; LREAL_ARR_D3[1, 2, 2] := 0.03125;
				LREAL_ARR_D3[2, 0, 0] := 0.015625; LREAL_ARR_D3[2, 0, 1] := 0.0078125; LREAL_ARR_D3[2, 0, 2] := 0.00390625;
				LREAL_ARR_D3[2, 1, 0] := 0.001953125; LREAL_ARR_D3[2, 1, 1] := 0.0009765625; LREAL_ARR_D3[2, 1, 2] := 0.00048828125;
				LREAL_ARR_D3[2, 2, 0] := 0.000244140625; LREAL_ARR_D3[2, 2, 1] := -1.0; LREAL_ARR_D3[2, 2, 2] := -0.5;
				iVarBinSize := ToAryByte(In:=LREAL_ARR_D3, Order:=_eBYTE_ORDER#_LOW_HIGH, AryOut:=iVarBin[0]);
				Inc(iVarIndex);
			133:
				iVarName := 'LREAL_ARR_D1_E1_LH';
				iVarDeclare := 'ARRAY[0..0] OF LREAL';
				iVarValue := '[1.0]';
				iVarKsType := 'nj::lreal_array_1d(1)';
				iVarKsId := 'lreal_arr_d1_e1_lh';
				
				Clear(LREAL_ARR_D1_E1);
				LREAL_ARR_D1_E1[0] := 1.0;
				iVarBinSize := ToAryByte(In:=LREAL_ARR_D1_E1, Order:=_eBYTE_ORDER#_LOW_HIGH, AryOut:=iVarBin[0]);
				Inc(iVarIndex);
			134:
				iVarName := 'LREAL_ARR_D2_E1_LH';
				iVarDeclare := 'ARRAY[0..0,0..0] OF LREAL';
				iVarValue := '[[1.0]]';
				iVarKsType := 'nj::lreal_array_2d(1,1)';
				iVarKsId := 'lreal_arr_d2_e1_lh';
				
				Clear(LREAL_ARR_D2_E1);
				LREAL_ARR_D2_E1[0, 0] := 1.0;
				iVarBinSize := ToAryByte(In:=LREAL_ARR_D2_E1, Order:=_eBYTE_ORDER#_LOW_HIGH, AryOut:=iVarBin[0]);
				Inc(iVarIndex);
			135:
				iVarName := 'LREAL_ARR_D3_E1_LH';
				iVarDeclare := 'ARRAY[0..0,0..0,0..0] OF LREAL';
				iVarValue := '[[[1.0]]]';
				iVarKsType := 'nj::lreal_array_3d(1,1,1)';
				iVarKsId := 'lreal_arr_d3_e1_lh';
				
				Clear(LREAL_ARR_D3_E1);
				LREAL_ARR_D3_E1[0, 0, 0] := 1.0;
				iVarBinSize := ToAryByte(In:=LREAL_ARR_D3_E1, Order:=_eBYTE_ORDER#_LOW_HIGH, AryOut:=iVarBin[0]);
				iVarIndex := iVarIndex - iVarIndex MOD 10 + 10;

			// STRING
			140:
				iVarName := 'STRING_N2_BY_TOARYBYTE_LH';
				iVarDeclare := 'STRING[2]';
				iVarValue := '"a"';
				iVarKsType := 'nj::string(2)';
				iVarKsId := 'string_n2_by_toarybyte_lh';

				Clear(STRING_N2);
				STRING_N2 := 'a';
				iVarBinSize := ToAryByte(In:=STRING_N2, Order:=_eBYTE_ORDER#_LOW_HIGH, AryOut:=iVarBin[0]);
				Inc(iVarIndex);
			141:
				iVarName := 'STRING_N2_BY_STRINGTOARY';
				iVarDeclare := 'STRING[2]';
				iVarValue := '"a"';

				Clear(STRING_N2);
				STRING_N2 := 'a';
				iVarBinSize := StringToAry(In:=STRING_N2, AryOut:=iVarBin[0]);
				Inc(iVarIndex);
			142:
				iVarName := 'STRING_N16_BY_TOARYBYTE_LH';
				iVarDeclare := 'STRING[16]';
				iVarValue := '"abc"';
				iVarKsType := 'nj::string(16)';
				iVarKsId := 'string_n16_by_toarybyte_lh';

				Clear(STRING_N16);
				STRING_N16 := 'abc';
				iVarBinSize := ToAryByte(In:=STRING_N16, Order:=_eBYTE_ORDER#_LOW_HIGH, AryOut:=iVarBin[0]);
				Inc(iVarIndex);
			143:
				iVarName := 'STRING_N16_BY_STRINGTOARY';
				iVarDeclare := 'STRING[16]';
				iVarValue := '"abc"';

				Clear(STRING_N16);
				STRING_N16 := 'abc';
				iVarBinSize := StringToAry(In:=STRING_N16, AryOut:=iVarBin[0]);
				Inc(iVarIndex);
			144:
				iVarName := 'STRING_2BYTE_CHAR_BY_TOARYBYTE_LH';
				iVarDeclare := 'STRING[16]';
				iVarValue := '"Σ-δ"';
				iVarKsType := 'nj::string(16)';
				iVarKsId := 'string_2byte_char_by_toarybyte_lh';

				Clear(STRING_N16);
				STRING_N16 := 'Σ-δ';
				iVarBinSize := ToAryByte(In:=STRING_N16, Order:=_eBYTE_ORDER#_LOW_HIGH, AryOut:=iVarBin[0]);
				Inc(iVarIndex);
			145:
				iVarName := 'STRING_2BYTE_CHAR_BY_STRINGTOARY';
				iVarDeclare := 'STRING[16]';
				iVarValue := '"Σ-δ"';

				Clear(STRING_N16);
				STRING_N16 := 'Σ-δ';
				iVarBinSize := StringToAry(In:=STRING_N16, AryOut:=iVarBin[0]);
				Inc(iVarIndex);
			146:
				iVarName := 'STRING_3BYTE_CHAR_BY_TOARYBYTE_LH';
				iVarDeclare := 'STRING[16]';
				iVarValue := '"ＪＰ"';
				iVarKsType := 'nj::string(16)';
				iVarKsId := 'string_3byte_char_by_toarybyte_lh';

				Clear(STRING_N16);
				STRING_N16 := 'ＪＰ';
				iVarBinSize := ToAryByte(In:=STRING_N16, Order:=_eBYTE_ORDER#_LOW_HIGH, AryOut:=iVarBin[0]);
				Inc(iVarIndex);
			147:
				iVarName := 'STRING_3BYTE_CHAR_BY_STRINGTOARY';
				iVarDeclare := 'STRING[16]';
				iVarValue := '"ＪＰ"';

				Clear(STRING_N16);
				STRING_N16 := 'ＪＰ';
				iVarBinSize := StringToAry(In:=STRING_N16, AryOut:=iVarBin[0]);
				Inc(iVarIndex);
			148:
				iVarName := 'STRING_4BYTE_CHAR_BY_TOARYBYTE_LH';
				iVarDeclare := 'STRING[16]';
				iVarValue := '"💯"';
				iVarKsType := 'nj::string(16)';
				iVarKsId := 'string_4byte_char_by_toarybyte_lh';

				Clear(STRING_N16);
				STRING_N16 := '💯';
				iVarBinSize := ToAryByte(In:=STRING_N16, Order:=_eBYTE_ORDER#_LOW_HIGH, AryOut:=iVarBin[0]);
				Inc(iVarIndex);
			149:
				iVarName := 'STRING_4BYTE_CHAR_BY_STRINGTOARY';
				iVarDeclare := 'STRING[16]';
				iVarValue := '"💯"';

				Clear(STRING_N16);
				STRING_N16 := '💯';
				iVarBinSize := StringToAry(In:=STRING_N16, AryOut:=iVarBin[0]);
				Inc(iVarIndex);

			// BOOL
			150:
				iVarName := 'BOOL_ARR_D1_LH';
				iVarDeclare := 'ARRAY[0..2] OF BOOL';
				iVarValue := '[true,false,true]';
				
				Clear(BOOL_ARR_D1);
				BOOL_ARR_D1[0] := TRUE; BOOL_ARR_D1[1] := FALSE; BOOL_ARR_D1[2] := TRUE;
				iVarBinSize := ToAryByte(In:=BOOL_ARR_D1, Order:=_eBYTE_ORDER#_LOW_HIGH, AryOut:=iVarBin[0]);
				Inc(iVarIndex);
			151:
				iVarName := 'BOOL_ARR_D2_LH';
				iVarDeclare := 'ARRAY[0..2,0..2] OF BOOL';
				iVarValue := '[[true,false,true], [false,true,false], [true,false,true]]';
				
				Clear(BOOL_ARR_D2);
				BOOL_ARR_D2[0, 0] := TRUE;  BOOL_ARR_D2[0, 1] := FALSE; BOOL_ARR_D2[0, 2] := TRUE;
				BOOL_ARR_D2[1, 0] := FALSE; BOOL_ARR_D2[1, 1] := TRUE;  BOOL_ARR_D2[1, 2] := FALSE;
				BOOL_ARR_D2[2, 0] := TRUE; BOOL_ARR_D2[2, 1] := FALSE;  BOOL_ARR_D2[2, 2] := TRUE;
				iVarBinSize := ToAryByte(In:=BOOL_ARR_D2, Order:=_eBYTE_ORDER#_LOW_HIGH, AryOut:=iVarBin[0]);
				Inc(iVarIndex);
			152:
				iVarName := 'BOOL_ARR_D3_LH';
				iVarDeclare := 'ARRAY[0..2,0..2,0..2] OF BOOL';
				iVarValue := '[[[true,false,true], [false,true,false], [true,false,true]],[[false,true,false], [true,false,true], [false,true,false]],[[true,false,true], [false,true,false], [true,false,true]]]';
				
				Clear(BOOL_ARR_D3);
				BOOL_ARR_D3[0, 0, 0] := TRUE;  BOOL_ARR_D3[0, 0, 1] := FALSE; BOOL_ARR_D3[0, 0, 2] := TRUE;
				BOOL_ARR_D3[0, 1, 0] := FALSE; BOOL_ARR_D3[0, 1, 1] := TRUE;  BOOL_ARR_D3[0, 1, 2] := FALSE;
				BOOL_ARR_D3[0, 2, 0] := TRUE;  BOOL_ARR_D3[0, 2, 1] := FALSE; BOOL_ARR_D3[0, 2, 2] := TRUE;
				BOOL_ARR_D3[1, 0, 0] := FALSE; BOOL_ARR_D3[1, 0, 1] := TRUE;  BOOL_ARR_D3[1, 0, 2] := FALSE;
				BOOL_ARR_D3[1, 1, 0] := TRUE;  BOOL_ARR_D3[1, 1, 1] := FALSE; BOOL_ARR_D3[1, 1, 2] := TRUE;
				BOOL_ARR_D3[1, 2, 0] := FALSE; BOOL_ARR_D3[1, 2, 1] := TRUE;  BOOL_ARR_D3[1, 2, 2] := FALSE;
				BOOL_ARR_D3[2, 0, 0] := TRUE;  BOOL_ARR_D3[2, 0, 1] := FALSE; BOOL_ARR_D3[2, 0, 2] := TRUE;
				BOOL_ARR_D3[2, 1, 0] := FALSE; BOOL_ARR_D3[2, 1, 1] := TRUE;  BOOL_ARR_D3[2, 1, 2] := FALSE;
				BOOL_ARR_D3[2, 2, 0] := TRUE;  BOOL_ARR_D3[2, 2, 1] := FALSE; BOOL_ARR_D3[2, 2, 2] := TRUE;
				
				iVarBinSize := ToAryByte(In:=BOOL_ARR_D3, Order:=_eBYTE_ORDER#_LOW_HIGH, AryOut:=iVarBin[0]);
				Inc(iVarIndex);
			153:
				iVarName := 'BOOL_ARR_D1_E1_LH';
				iVarDeclare := 'ARRAY[0..0] OF BOOL';
				iVarValue := '[true]';
				
				Clear(BOOL_ARR_D1_E1);
				BOOL_ARR_D1_E1[0] := TRUE;
				iVarBinSize := ToAryByte(In:=BOOL_ARR_D1_E1, Order:=_eBYTE_ORDER#_LOW_HIGH, AryOut:=iVarBin[0]);
				Inc(iVarIndex);
			154:
				iVarName := 'BOOL_ARR_D2_E1_LH';
				iVarDeclare := 'ARRAY[0..0,0..0] OF BOOL';
				iVarValue := '[[true]]';
				
				Clear(BOOL_ARR_D2_E1);
				BOOL_ARR_D2_E1[0, 0] := TRUE;
				iVarBinSize := ToAryByte(In:=BOOL_ARR_D2_E1, Order:=_eBYTE_ORDER#_LOW_HIGH, AryOut:=iVarBin[0]);
				Inc(iVarIndex);
			155:
				iVarName := 'BOOL_ARR_D3_E1_LH';
				iVarDeclare := 'ARRAY[0..0,0..0,0..0] OF BOOL';
				iVarValue := '[[[true]]]';
				
				Clear(BOOL_ARR_D3_E1);
				BOOL_ARR_D3_E1[0, 0, 0] := TRUE;
				iVarBinSize := ToAryByte(In:=BOOL_ARR_D3_E1, Order:=_eBYTE_ORDER#_LOW_HIGH, AryOut:=iVarBin[0]);
				iVarIndex := iVarIndex - iVarIndex MOD 10 + 10;
			
			// TIME
			160:
				iVarName := 'TIME_ARR_D1_LH';
				iVarDeclare := 'ARRAY[0..2] OF TIME';
				// iVarValue := '["00:00:00","00:00:00.0000001","106751.23:47:16.8547758"]';
				iVarValue := '[0,100,9223372036854775800]';
				iVarKsType := 'nj::time_array_1d(3)';
				iVarKsId := 'time_arr_d1_lh';
				
				Clear(TIME_ARR_D1);
				TIME_ARR_D1[0] := TIME#0s;
				TIME_ARR_D1[1] := TIME#0.0001ms;
				TIME_ARR_D1[2] := TIME#106751d_23h_47m_16s_854.7758ms;
				iVarBinSize := ToAryByte(In:=TIME_ARR_D1, Order:=_eBYTE_ORDER#_LOW_HIGH, AryOut:=iVarBin[0]);
				Inc(iVarIndex);
			161:
				iVarName := 'TIME_ARR_D2_LH';
				iVarDeclare := 'ARRAY[0..2,0..2] OF TIME';
				// iVarValue := '[["00:00:00","00:00:00.0000001","106751.23:47:16.8547758"],["00:00:00.000001","00:00:00.1","00:01:00"],["01:00:00.0000001","1.00:00:00","-00:00:00.0000001"]]';
				iVarValue := '[[0,100,9223372036854775800],[1000,1000000,60000000000],[3600000000000,86400000000000,-100]]';
				iVarKsType := 'nj::time_array_2d(3,3)';
				iVarKsId := 'time_arr_d2_lh';
				
				Clear(TIME_ARR_D2);
				TIME_ARR_D2[0, 0] := TIME#0s;
				TIME_ARR_D2[0, 1] := TIME#0.0001ms;
				TIME_ARR_D2[0, 2] := TIME#106751d_23h_47m_16s_854.7758ms;
				TIME_ARR_D2[1, 0] := TIME#0.001ms;
				TIME_ARR_D2[1, 1] := TIME#1ms;
				TIME_ARR_D2[1, 2] := TIME#1m;
				TIME_ARR_D2[2, 0] := TIME#1h;
				TIME_ARR_D2[2, 1] := TIME#1d;
				TIME_ARR_D2[2, 2] := TIME#-0.0001ms;
				iVarBinSize := ToAryByte(In:=TIME_ARR_D2, Order:=_eBYTE_ORDER#_LOW_HIGH, AryOut:=iVarBin[0]);
				Inc(iVarIndex);
			162:
				iVarName := 'TIME_ARR_D3_LH';
				iVarDeclare := 'ARRAY[0..2,0..2,0..2] OF TIME';
				// iVarValue := '[[["00:00:00","00:00:00.0000001","106751.23:47:16.8547758"],["00:00:00.000001","00:00:00.1","00:01:00"],["01:00:00.0000001","1.00:00:00","-00:00:00.0000001"]], [["-106751.23:47:16.8547758","-00:00:00.000001","-00:00:00.1"],["-00:01:00","-01:00:00.0000001","-1.00:00:00"],["00:00:00.0009999","00:00:00.999","00:00:59"]], [["00:59:00","23:00:00","99999.00:00:00"],["-00:00:00.0009999","-00:00:00.999","-00:00:59"],["-00:59:00","-23:00:00","-99999.00:00:00"]]]';
				iVarValue := '[[[0,100,9223372036854775800],[1000,1000000,60000000000],[3600000000000,86400000000000,-100]],[[-9223372036854775800,-1000,-1000000],[-60000000000,-3600000000000,-86400000000000],[999900,999000000,59000000000]],[[3540000000000,82800000000000,8639913600000000000],[-999900,-999000000,-59000000000],[-3540000000000,-82800000000000,-8639913600000000000]]]';
				iVarKsType := 'nj::time_array_3d(3,3,3)';
				iVarKsId := 'time_arr_d3_lh';
				
				Clear(TIME_ARR_D3);
				TIME_ARR_D3[0, 0, 0] := TIME#0s;
				TIME_ARR_D3[0, 0, 1] := TIME#0.0001ms;
				TIME_ARR_D3[0, 0, 2] := TIME#106751d_23h_47m_16s_854.7758ms;
				TIME_ARR_D3[0, 1, 0] := TIME#0.001ms;
				TIME_ARR_D3[0, 1, 1] := TIME#1ms;
				TIME_ARR_D3[0, 1, 2] := TIME#1m;
				TIME_ARR_D3[0, 2, 0] := TIME#1h;
				TIME_ARR_D3[0, 2, 1] := TIME#1d;
				TIME_ARR_D3[0, 2, 2] := TIME#-0.0001ms;
				
				TIME_ARR_D3[1, 0, 0] := TIME#-106751d_23h_47m_16s_854.7758ms;
				TIME_ARR_D3[1, 0, 1] := TIME#-0.001ms;
				TIME_ARR_D3[1, 0, 2] := TIME#-1ms;
				TIME_ARR_D3[1, 1, 0] := TIME#-1m;
				TIME_ARR_D3[1, 1, 1] := TIME#-1h;
				TIME_ARR_D3[1, 1, 2] := TIME#-1d;
				TIME_ARR_D3[1, 2, 0] := TIME#0.9999ms;
				TIME_ARR_D3[1, 2, 1] := TIME#999ms;
				TIME_ARR_D3[1, 2, 2] := TIME#59s;

				TIME_ARR_D3[2, 0, 0] := TIME#59m;
				TIME_ARR_D3[2, 0, 1] := TIME#23h;
				TIME_ARR_D3[2, 0, 2] := TIME#99999d;
				TIME_ARR_D3[2, 1, 0] := TIME#-0.9999ms;
				TIME_ARR_D3[2, 1, 1] := TIME#-999ms;
				TIME_ARR_D3[2, 1, 2] := TIME#-59s;
				TIME_ARR_D3[2, 2, 0] := TIME#-59m;
				TIME_ARR_D3[2, 2, 1] := TIME#-23h;
				TIME_ARR_D3[2, 2, 2] := TIME#-99999d;
				iVarBinSize := ToAryByte(In:=TIME_ARR_D3, Order:=_eBYTE_ORDER#_LOW_HIGH, AryOut:=iVarBin[0]);
				Inc(iVarIndex);
			163:
				iVarName := 'TIME_ARR_D1_E1_LH';
				iVarDeclare := 'ARRAY[0..0] OF TIME';
				// iVarValue := '["00:00:00.0000001"]';
				iVarValue := '[100]';
				iVarKsType := 'nj::time_array_1d(1)';
				iVarKsId := 'time_arr_d1_e1_lh';
				
				Clear(TIME_ARR_D1_E1);
				TIME_ARR_D1_E1[0] := TIME#0.0001ms;
				iVarBinSize := ToAryByte(In:=TIME_ARR_D1_E1, Order:=_eBYTE_ORDER#_LOW_HIGH, AryOut:=iVarBin[0]);
				Inc(iVarIndex);
			164:
				iVarName := 'TOD_ARR_D2_E1_LH';
				iVarDeclare := 'ARRAY[0..0,0..0] OF TIME';
				// iVarValue := '[["00:00:00.0000001"]]';
				iVarValue := '[[100]]';
				iVarKsType := 'nj::time_array_2d(1,1)';
				iVarKsId := 'time_arr_d2_e1_lh';
				
				Clear(TIME_ARR_D2_E1);
				TIME_ARR_D2_E1[0, 0] := TIME#0.0001ms;
				iVarBinSize := ToAryByte(In:=TIME_ARR_D2_E1, Order:=_eBYTE_ORDER#_LOW_HIGH, AryOut:=iVarBin[0]);
				Inc(iVarIndex);
			165:
				iVarName := 'TIME_ARR_D3_E1_LH';
				iVarDeclare := 'ARRAY[0..0,0..0,0..0] OF TIME';
				// iVarValue := '[[["00:00:00.0000001"]]]';
				iVarValue := '[[[100]]]';
				iVarKsType := 'nj::time_array_3d(1,1,1)';
				iVarKsId := 'time_arr_d3_e1_lh';
				
				Clear(TIME_ARR_D3_E1);
				TIME_ARR_D3_E1[0, 0, 0] := TIME#0.0001ms;
				iVarBinSize := ToAryByte(In:=TIME_ARR_D3_E1, Order:=_eBYTE_ORDER#_LOW_HIGH, AryOut:=iVarBin[0]);
				iVarIndex := iVarIndex - iVarIndex MOD 10 + 10;

			// DATE
			170:
				iVarName := 'DATE_ARR_D1_LH';
				iVarDeclare := 'ARRAY[0..2] OF DATE';
				// iVarValue := '["1970-01-01", "1970-01-02", "2026-06-04"]';
				iVarValue := '[0, 86400000000000,1780531200000000000]';
				iVarKsType := 'nj::date_array_1d(3)';
				iVarKsId := 'date_arr_d1_lh';
				
				Clear(DATE_ARR_D1);
				DATE_ARR_D1[0] := DATE#1970-01-01;
				DATE_ARR_D1[1] := DATE#1970-01-02;
				DATE_ARR_D1[2] := DATE#2026-06-04;
				iVarBinSize := ToAryByte(In:=DATE_ARR_D1, Order:=_eBYTE_ORDER#_LOW_HIGH, AryOut:=iVarBin[0]);
				Inc(iVarIndex);
			171:
				iVarName := 'DATE_ARR_D2_LH';
				iVarDeclare := 'ARRAY[0..2,0..2] OF DATE';
				// iVarValue := '[["1970-01-01", "1970-01-10", "1970-02-01"], ["1970-10-01", "1971-01-01", "1980-01-01"], ["2070-01-01", "1970-01-31", "1970-12-01"]]';
				iVarValue := '[[0,777600000000000,2678400000000000],[23587200000000000,31536000000000000,315532800000000000],[3155760000000000000,2592000000000000,28857600000000000]]';
				iVarKsType := 'nj::date_array_2d(3,3)';
				iVarKsId := 'date_arr_d2_lh';
				
				Clear(DATE_ARR_D2);
				DATE_ARR_D2[0, 0] := DATE#1970-01-01;
				DATE_ARR_D2[0, 1] := DATE#1970-01-10;
				DATE_ARR_D2[0, 2] := DATE#1970-02-01;
				DATE_ARR_D2[1, 0] := DATE#1970-10-01;
				DATE_ARR_D2[1, 1] := DATE#1971-01-01;
				DATE_ARR_D2[1, 2] := DATE#1980-01-01;
				DATE_ARR_D2[2, 0] := DATE#2070-01-01;
				DATE_ARR_D2[2, 1] := DATE#1970-01-31;
				DATE_ARR_D2[2, 2] := DATE#1970-12-01;
				iVarBinSize := ToAryByte(In:=DATE_ARR_D2, Order:=_eBYTE_ORDER#_LOW_HIGH, AryOut:=iVarBin[0]);
				Inc(iVarIndex);
			172:
				iVarName := 'DATE_ARR_D3_LH';
				iVarDeclare := 'ARRAY[0..2,0..2,0..2] OF DATE';
				// iVarValue := '[[["1970-01-01","1970-01-10","1970-02-01"],["1970-10-01","1971-01-01","1980-01-01"],["2070-01-01","1970-01-31","1970-12-01"]],[["2106-01-01","2106-02-06","1999-12-31"],["2000-01-01","2000-01-02","2036-02-06"],["2036-02-07","2036-02-08","1970-12-31"]],[["1971-11-15","1977-05-25","1989-11-09"],["1991-12-25","1995-08-24","1997-05-11"],["2007-01-09","2008-10-31","2022-11-30"]]]';
				iVarValue := '[[[0,777600000000000,2678400000000000],[23587200000000000,31536000000000000,315532800000000000],[3155760000000000000,2592000000000000,28857600000000000]],[[4291747200000000000,4294857600000000000,946598400000000000],[946684800000000000,946771200000000000,2085868800000000000],[2085955200000000000,2086041600000000000,31449600000000000]],[[59011200000000000,233366400000000000,626572800000000000],[693619200000000000,809222400000000000,863308800000000000],[1168300800000000000,1225411200000000000,1669766400000000000]]]';
				iVarKsType := 'nj::date_array_3d(3,3,3)';
				iVarKsId := 'date_arr_d3_lh';
				
				Clear(DATE_ARR_D3);
				DATE_ARR_D3[0, 0, 0] := DATE#1970-01-01;
				DATE_ARR_D3[0, 0, 1] := DATE#1970-01-10;
				DATE_ARR_D3[0, 0, 2] := DATE#1970-02-01;
				DATE_ARR_D3[0, 1, 0] := DATE#1970-10-01;
				DATE_ARR_D3[0, 1, 1] := DATE#1971-01-01;
				DATE_ARR_D3[0, 1, 2] := DATE#1980-01-01;
				DATE_ARR_D3[0, 2, 0] := DATE#2070-01-01;
				DATE_ARR_D3[0, 2, 1] := DATE#1970-01-31;
				DATE_ARR_D3[0, 2, 2] := DATE#1970-12-01;

				DATE_ARR_D3[1, 0, 0] := DATE#2106-01-01;
				DATE_ARR_D3[1, 0, 1] := DATE#2106-02-06;
				DATE_ARR_D3[1, 0, 2] := DATE#1999-12-31;
				DATE_ARR_D3[1, 1, 0] := DATE#2000-01-01;
				DATE_ARR_D3[1, 1, 1] := DATE#2000-01-02;
				DATE_ARR_D3[1, 1, 2] := DATE#2036-02-06;
				DATE_ARR_D3[1, 2, 0] := DATE#2036-02-07;
				DATE_ARR_D3[1, 2, 1] := DATE#2036-02-08;
				DATE_ARR_D3[1, 2, 2] := DATE#1970-12-31;
				
				DATE_ARR_D3[2, 0, 0] := DATE#1971-11-15;
				DATE_ARR_D3[2, 0, 1] := DATE#1977-05-25;
				DATE_ARR_D3[2, 0, 2] := DATE#1989-11-09;
				DATE_ARR_D3[2, 1, 0] := DATE#1991-12-25;
				DATE_ARR_D3[2, 1, 1] := DATE#1995-08-24;
				DATE_ARR_D3[2, 1, 2] := DATE#1997-05-11;
				DATE_ARR_D3[2, 2, 0] := DATE#2007-01-09;
				DATE_ARR_D3[2, 2, 1] := DATE#2008-10-31;
				DATE_ARR_D3[2, 2, 2] := DATE#2022-11-30;

				iVarBinSize := ToAryByte(In:=DATE_ARR_D3, Order:=_eBYTE_ORDER#_LOW_HIGH, AryOut:=iVarBin[0]);
				Inc(iVarIndex);
			173:
				iVarName := 'DATE_ARR_D1_E1_LH';
				iVarDeclare := 'ARRAY[0..0] OF DATE';
				// iVarValue := '["1970-01-02"]';
				iVarValue := '[86400000000000]';
				iVarKsType := 'nj::date_array_1d(1)';
				iVarKsId := 'date_arr_d1_e1_lh';
				
				Clear(DATE_ARR_D1_E1);
				DATE_ARR_D1_E1[0] := DATE#1970-01-02;
				iVarBinSize := ToAryByte(In:=DATE_ARR_D1_E1, Order:=_eBYTE_ORDER#_LOW_HIGH, AryOut:=iVarBin[0]);
				Inc(iVarIndex);
			174:
				iVarName := 'DATE_ARR_D2_E1_LH';
				iVarDeclare := 'ARRAY[0..0,0..0] OF DATE';
				// iVarValue := '[["1970-01-02"]]';
				iVarValue := '[[86400000000000]]';
				iVarKsType := 'nj::date_array_2d(1,1)';
				iVarKsId := 'date_arr_d2_e1_lh';
				
				Clear(DATE_ARR_D2_E1);
				DATE_ARR_D2_E1[0, 0] := DATE#1970-01-02;
				iVarBinSize := ToAryByte(In:=DATE_ARR_D2_E1, Order:=_eBYTE_ORDER#_LOW_HIGH, AryOut:=iVarBin[0]);
				Inc(iVarIndex);
			175:
				iVarName := 'DATE_ARR_D3_E1_LH';
				iVarDeclare := 'ARRAY[0..0,0..0,0..0] OF DATE';
				// iVarValue := '[[["1970-01-02"]]]';
				iVarValue := '[[[86400000000000]]]';
				iVarKsType := 'nj::date_array_3d(1,1,1)';
				iVarKsId := 'date_arr_d3_e1_lh';
				
				Clear(DATE_ARR_D3_E1);
				DATE_ARR_D3_E1[0, 0, 0] := DATE#1970-01-02;
				iVarBinSize := ToAryByte(In:=DATE_ARR_D3_E1, Order:=_eBYTE_ORDER#_LOW_HIGH, AryOut:=iVarBin[0]);
				iVarIndex := iVarIndex - iVarIndex MOD 10 + 10;
			
			// TIME_OF_DAY
			180:
				iVarName := 'TOD_ARR_D1_LH';
				iVarDeclare := 'ARRAY[0..2] OF TIME_OF_DAY';
				// iVarValue := '["00:00:00.0000000", "00:00:00.0000001", "23:59:59.9999999"]';
				iVarValue := '[0,100,86399999999900]';
				iVarKsType := 'nj::time_of_day_array_1d(3)';
				iVarKsId := 'time_of_day_arr_d1_lh';
				
				Clear(TOD_ARR_D1);
				TOD_ARR_D1[0] := TOD#00:00:00.000000000;
				TOD_ARR_D1[1] := TOD#00:00:00.000000100;
				TOD_ARR_D1[2] := TOD#23:59:59.999999900;
				iVarBinSize := ToAryByte(In:=TOD_ARR_D1, Order:=_eBYTE_ORDER#_LOW_HIGH, AryOut:=iVarBin[0]);
				Inc(iVarIndex);
			181:
				iVarName := 'TOD_ARR_D2_LH';
				iVarDeclare := 'ARRAY[0..2,0..2] OF TIME_OF_DAY';
				// iVarValue := '[["00:00:00.0000000", "00:00:00.0000001", "00:00:00.0000010"], ["00:00:00.0010000", "01:00:01.0000000", "00:00:10.0000000"], ["00:01:00.0000000", "00:10:00.0000000", "01:00:00.0000000"]]';
				iVarValue := '[[0,100,1000],[100000,1000000000,10000000000],[60000000000,600000000000,3600000000000]]';
				iVarKsType := 'nj::time_of_day_array_2d(3,3)';
				iVarKsId := 'time_of_day_arr_d2_lh';
				
				Clear(TOD_ARR_D2);
				TOD_ARR_D2[0, 0] := TOD#00:00:00.000000000;
				TOD_ARR_D2[0, 1] := TOD#00:00:00.000000100;
				TOD_ARR_D2[0, 2] := TOD#00:00:00.000001000;
				TOD_ARR_D2[1, 0] := TOD#00:00:00.000100000;
				TOD_ARR_D2[1, 1] := TOD#00:00:01.000000000;
				TOD_ARR_D2[1, 2] := TOD#00:00:10.000000000;
				TOD_ARR_D2[2, 0] := TOD#00:01:00.000000000;
				TOD_ARR_D2[2, 1] := TOD#00:10:00.000000000;
				TOD_ARR_D2[2, 2] := TOD#01:00:00.000000000;
				iVarBinSize := ToAryByte(In:=TOD_ARR_D2, Order:=_eBYTE_ORDER#_LOW_HIGH, AryOut:=iVarBin[0]);
				Inc(iVarIndex);
			182:
				iVarName := 'TOD_ARR_D3_LH';
				iVarDeclare := 'ARRAY[0..2,0..2,0..2] OF TIME_OF_DAY';
				// iVarValue := '[[["00:00:00.0000000","00:00:00.0000001","00:00:00.0000010"],["00:00:00.0010000","00:00:01.0000000","00:00:10.0000000"],["00:01:00.0000000","00:10:00.0000000","01:00:00.0000000"]], [["10:00:00.0000000","00:00:00.9999999","00:00:09.0000000"],["00:00:59.0000000","00:09:00.0000000","00:59:00.0000000"],["09:00:00.0000000","23:00:00.0000000","00:00:09.9999999"]], [["00:00:59.9999999","00:09:59.9999999","00:59:59.9999999"],["09:59:59.9999999","23:59:59.9999999","11:59:59.9999999"],["12:00:00.0000000","12:00:00.0000001","12:00:00.0010000"]]]';
				iVarValue := '[[[0,100,1000],[1000000,1000000000,10000000000],[60000000000,600000000000,3600000000000]],[[36000000000000,999999900,9000000000],[59000000000,540000000000,3540000000000],[32400000000000,82800000000000,9999999900]],[[59999999900,599999999900,3599999999900],[35999999999900,86399999999900,43199999999900],[43200000000000,43200000000100,43200001000000]]]';
				iVarKsType := 'nj::time_of_day_array_3d(3,3,3)';
				iVarKsId := 'time_of_day_arr_d3_lh';
				
				Clear(TOD_ARR_D3);
				TOD_ARR_D3[0, 0, 0] := TOD#00:00:00.000000000;
				TOD_ARR_D3[0, 0, 1] := TOD#00:00:00.000000100;
				TOD_ARR_D3[0, 0, 2] := TOD#00:00:00.000001000;
				TOD_ARR_D3[0, 1, 0] := TOD#00:00:00.001000000;
				TOD_ARR_D3[0, 1, 1] := TOD#00:00:01.000000000;
				TOD_ARR_D3[0, 1, 2] := TOD#00:00:10.000000000;
				TOD_ARR_D3[0, 2, 0] := TOD#00:01:00.000000000;
				TOD_ARR_D3[0, 2, 1] := TOD#00:10:00.000000000;
				TOD_ARR_D3[0, 2, 2] := TOD#01:00:00.000000000;

				TOD_ARR_D3[1, 0, 0] := TOD#10:00:00.000000000;
				TOD_ARR_D3[1, 0, 1] := TOD#00:00:00.999999900;
				TOD_ARR_D3[1, 0, 2] := TOD#00:00:09.000000000;
				TOD_ARR_D3[1, 1, 0] := TOD#00:00:59.000000000;
				TOD_ARR_D3[1, 1, 1] := TOD#00:09:00.000000000;
				TOD_ARR_D3[1, 1, 2] := TOD#00:59:00.000000000;
				TOD_ARR_D3[1, 2, 0] := TOD#09:00:00.000000000;
				TOD_ARR_D3[1, 2, 1] := TOD#23:00:00.000000000;
				TOD_ARR_D3[1, 2, 2] := TOD#00:00:09.999999900;
				
				TOD_ARR_D3[2, 0, 0] := TOD#00:00:59.999999900;
				TOD_ARR_D3[2, 0, 1] := TOD#00:09:59.999999900;
				TOD_ARR_D3[2, 0, 2] := TOD#00:59:59.999999900;
				TOD_ARR_D3[2, 1, 0] := TOD#09:59:59.999999900;
				TOD_ARR_D3[2, 1, 1] := TOD#23:59:59.999999900;
				TOD_ARR_D3[2, 1, 2] := TOD#11:59:59.999999900;
				TOD_ARR_D3[2, 2, 0] := TOD#12:00:00.000000000;
				TOD_ARR_D3[2, 2, 1] := TOD#12:00:00.000000100;
				TOD_ARR_D3[2, 2, 2] := TOD#12:00:00.001000000;
				iVarBinSize := ToAryByte(In:=TOD_ARR_D3, Order:=_eBYTE_ORDER#_LOW_HIGH, AryOut:=iVarBin[0]);
				Inc(iVarIndex);
			183:
				iVarName := 'TOD_ARR_D1_E1_LH';
				iVarDeclare := 'ARRAY[0..0] OF TIME_OF_DAY';
				// iVarValue := '["00:00:00.0000001"]';
				iVarValue := '[100]';
				iVarKsType := 'nj::time_of_day_array_1d(1)';
				iVarKsId := 'time_of_day_arr_d1_e1_lh';
				
				Clear(TOD_ARR_D1_E1);
				TOD_ARR_D1_E1[0] := TOD#00:00:00.000000100;
				iVarBinSize := ToAryByte(In:=TOD_ARR_D1_E1, Order:=_eBYTE_ORDER#_LOW_HIGH, AryOut:=iVarBin[0]);
				Inc(iVarIndex);
			184:
				iVarName := 'TOD_ARR_D2_E1_LH';
				iVarDeclare := 'ARRAY[0..0,0..0] OF TIME_OF_DAY';
				// iVarValue := '[["00:00:00.0000001"]]';
				iVarValue := '[[100]]';
				iVarKsType := 'nj::time_of_day_array_2d(1,1)';
				iVarKsId := 'time_of_day_arr_d2_e1_lh';
				
				Clear(TOD_ARR_D2_E1);
				TOD_ARR_D2_E1[0, 0] := TOD#00:00:00.000000100;
				iVarBinSize := ToAryByte(In:=TOD_ARR_D2_E1, Order:=_eBYTE_ORDER#_LOW_HIGH, AryOut:=iVarBin[0]);
				Inc(iVarIndex);
			185:
				iVarName := 'TOD_ARR_D3_E1_LH';
				iVarDeclare := 'ARRAY[0..0,0..0,0..0] OF TIME_OF_DAY';
				// iVarValue := '[[["00:00:00.0000001"]]]';
				iVarValue := '[[[100]]]';
				iVarKsType := 'nj::time_of_day_array_3d(1,1,1)';
				iVarKsId := 'time_of_day_arr_d3_e1_lh';
				
				Clear(TOD_ARR_D3_E1);
				TOD_ARR_D3_E1[0, 0, 0] := TOD#00:00:00.000000100;
				iVarBinSize := ToAryByte(In:=TOD_ARR_D3_E1, Order:=_eBYTE_ORDER#_LOW_HIGH, AryOut:=iVarBin[0]);
				iVarIndex := iVarIndex - iVarIndex MOD 10 + 10;

			// DATE_AND_TIME
			190:
				iVarName := 'DT_ARR_D1_LH';
				iVarDeclare := 'ARRAY[0..2] OF DATE_AND_TIME';
				// iVarValue := '["1970-01-01T00:00:00.0000000Z", "1970-01-01T00:00:00.0000001Z", "2026-06-04T09:00:00.0000000Z"]';
				iVarValue := '[0,100,1780563600000000000]';
				iVarKsType := 'nj::date_and_time_array_1d(3)';
				iVarKsId := 'date_and_time_arr_d1_lh';

				Clear(DT_ARR_D1);
				DT_ARR_D1[0] := DT#1970-01-01-00:00:00.000000000;
				DT_ARR_D1[1] := DT#1970-01-01-00:00:00.000000100;
				DT_ARR_D1[2] := DT#2026-06-04-09:00:00.000000000;
				iVarBinSize := ToAryByte(In:=DT_ARR_D1, Order:=_eBYTE_ORDER#_LOW_HIGH, AryOut:=iVarBin[0]);
				Inc(iVarIndex);
			191:
				iVarName := 'DT_ARR_D2_LH';
				iVarDeclare := 'ARRAY[0..2,0..2] OF DATE_AND_TIME';
				// iVarValue := '[["1970-01-01T00:00:00.0000000Z", "1970-01-01T00:00:00.0000001Z", "1970-01-01T00:00:00.0000010Z"], ["1970-01-01T00:00:00.0010000Z", "1970-01-01T01:00:01.0000000Z", "1970-01-01T00:00:10.0000000Z"], ["1970-01-01T00:01:00.0000000Z", "1970-01-01T00:10:00.0000000Z", "1970-01-01T01:00:00.0000000Z"]]';
				iVarValue := '[[0,100,1000],[100000,1000000000,10000000000],[60000000000,600000000000,3600000000000]]';
				iVarKsType := 'nj::date_and_time_array_2d(3,3)';
				iVarKsId := 'date_and_time_arr_d2_lh';
				
				Clear(DT_ARR_D2);
				DT_ARR_D2[0, 0] := DT#1970-01-01-00:00:00.000000000;
				DT_ARR_D2[0, 1] := DT#1970-01-01-00:00:00.000000100;
				DT_ARR_D2[0, 2] := DT#1970-01-01-00:00:00.000001000;
				DT_ARR_D2[1, 0] := DT#1970-01-01-00:00:00.000100000;
				DT_ARR_D2[1, 1] := DT#1970-01-01-00:00:01.000000000;
				DT_ARR_D2[1, 2] := DT#1970-01-01-00:00:10.000000000;
				DT_ARR_D2[2, 0] := DT#1970-01-01-00:01:00.000000000;
				DT_ARR_D2[2, 1] := DT#1970-01-01-00:10:00.000000000;
				DT_ARR_D2[2, 2] := DT#1970-01-01-01:00:00.000000000;
				iVarBinSize := ToAryByte(In:=DT_ARR_D2, Order:=_eBYTE_ORDER#_LOW_HIGH, AryOut:=iVarBin[0]);
				Inc(iVarIndex);
			192:
				iVarName := 'DT_ARR_D3_LH';
				iVarDeclare := 'ARRAY[0..2,0..2,0..2] OF DATE_AND_TIME';
				// iVarValue := '[[["1970-01-01T00:00:00.0000000Z", "1970-01-01T00:00:00.0000001Z", "1970-01-01T00:00:00.0000010Z"], ["1970-01-01T00:00:00.0010000Z", "1970-01-01T01:00:01.0000000Z", "1970-01-01T00:00:10.0000000Z"], ["1970-01-01T00:01:00.0000000Z", "1970-01-01T00:10:00.0000000Z", "1970-01-01T01:00:00.0000000Z"]], [["1970-01-01T10:00:00.0000000Z", "1970-01-02T00:00:00.0000000Z", "1970-01-10T00:00:00.0000000Z"], ["1970-02-01T00:00:00.0000000Z", "1970-10-01T00:00:00.0000000Z", "1971-01-01T00:00:00.0000000Z"], ["1980-01-01T00:00:00.0000000Z", "2070-01-01T00:00:00.0000000Z", "1970-01-01T00:00:00.9999999Z"]], [["1970-01-01T00:00:09.9999999Z", "1970-01-01T00:00:59.9999999Z", "1970-01-01T00:09:59.9999999Z"], ["1970-01-01T00:59:59.9999999Z", "1970-01-01T09:59:59.9999999Z", "1970-01-01T23:59:59.9999999Z"], ["1970-01-09T23:59:59.9999999Z", "1970-01-31T23:59:59.9999999Z", "1970-09-30T23:59:59.9999999Z"]]]';
				iVarValue := '[[[0,100,1000],[1000000,1000000000,10000000000],[60000000000,600000000000,3600000000000]],[[36000000000000,86400000000000,777600000000000],[2678400000000000,23587200000000000,31536000000000000],[315532800000000000,3155760000000000000,999999900]],[[9999999900,59999999900,599999999900],[3599999999900,35999999999900,86399999999900],[777599999999900,2678399999999900,23587199999999900]]]';
				iVarKsType := 'nj::date_and_time_array_3d(3,3,3)';
				iVarKsId := 'date_and_time_arr_d3_lh';
				
				Clear(DT_ARR_D3);
				DT_ARR_D3[0, 0, 0] := DT#1970-01-01-00:00:00.000000000;
				DT_ARR_D3[0, 0, 1] := DT#1970-01-01-00:00:00.000000100;
				DT_ARR_D3[0, 0, 2] := DT#1970-01-01-00:00:00.000001000;
				DT_ARR_D3[0, 1, 0] := DT#1970-01-01-00:00:00.001000000;
				DT_ARR_D3[0, 1, 1] := DT#1970-01-01-00:00:01.000000000;
				DT_ARR_D3[0, 1, 2] := DT#1970-01-01-00:00:10.000000000;
				DT_ARR_D3[0, 2, 0] := DT#1970-01-01-00:01:00.000000000;
				DT_ARR_D3[0, 2, 1] := DT#1970-01-01-00:10:00.000000000;
				DT_ARR_D3[0, 2, 2] := DT#1970-01-01-01:00:00.000000000;

				DT_ARR_D3[1, 0, 0] := DT#1970-01-01-10:00:00.000000000;
				DT_ARR_D3[1, 0, 1] := DT#1970-01-02-00:00:00.000000000;
				DT_ARR_D3[1, 0, 2] := DT#1970-01-10-00:00:00.000000000;
				DT_ARR_D3[1, 1, 0] := DT#1970-02-01-00:00:00.000000000;
				DT_ARR_D3[1, 1, 1] := DT#1970-10-01-00:00:00.000000000;
				DT_ARR_D3[1, 1, 2] := DT#1971-01-01-00:00:00.000000000;
				DT_ARR_D3[1, 2, 0] := DT#1980-01-01-00:00:00.000000000;
				DT_ARR_D3[1, 2, 1] := DT#2070-01-01-00:00:00.000000000;
				DT_ARR_D3[1, 2, 2] := DT#1970-01-01-00:00:00.999999900;

				DT_ARR_D3[2, 0, 0] := DT#1970-01-01-00:00:09.999999900;
				DT_ARR_D3[2, 0, 1] := DT#1970-01-01-00:00:59.999999900;
				DT_ARR_D3[2, 0, 2] := DT#1970-01-01-00:09:59.999999900;
				DT_ARR_D3[2, 1, 0] := DT#1970-01-01-00:59:59.999999900;
				DT_ARR_D3[2, 1, 1] := DT#1970-01-01-09:59:59.999999900;
				DT_ARR_D3[2, 1, 2] := DT#1970-01-01-23:59:59.999999900;
				DT_ARR_D3[2, 2, 0] := DT#1970-01-09-23:59:59.999999900;
				DT_ARR_D3[2, 2, 1] := DT#1970-01-31-23:59:59.999999900;
				DT_ARR_D3[2, 2, 2] := DT#1970-09-30-23:59:59.999999900;

				iVarBinSize := ToAryByte(In:=DT_ARR_D3, Order:=_eBYTE_ORDER#_LOW_HIGH, AryOut:=iVarBin[0]);
				Inc(iVarIndex);
			193:
				iVarName := 'DT_ARR_D1_E1_LH';
				iVarDeclare := 'ARRAY[0..0] OF DATE_AND_TIME';
				// iVarValue := '["1970-01-01T00:00:00.0000001Z"]';
				iVarValue := '[100]';
				iVarKsType := 'nj::date_and_time_array_1d(1)';
				iVarKsId := 'date_and_time_arr_d1_e1_lh';
				
				Clear(DT_ARR_D1_E1);
				DT_ARR_D1_E1[0] := DT#1970-01-01-00:00:00.000000100;
				iVarBinSize := ToAryByte(In:=DT_ARR_D1_E1, Order:=_eBYTE_ORDER#_LOW_HIGH, AryOut:=iVarBin[0]);
				Inc(iVarIndex);
			194:
				iVarName := 'DT_ARR_D2_E1_LH';
				iVarDeclare := 'ARRAY[0..0,0..0] OF DATE_AND_TIME';
				// iVarValue := '[["1970-01-01T00:00:00.0000001Z"]]';
				iVarValue := '[[100]]';
				iVarKsType := 'nj::date_and_time_array_2d(1,1)';
				iVarKsId := 'date_and_time_arr_d2_e1_lh';
				
				Clear(DT_ARR_D2_E1);
				DT_ARR_D2_E1[0, 0] := DT#1970-01-01-00:00:00.000000100;
				iVarBinSize := ToAryByte(In:=DT_ARR_D2_E1, Order:=_eBYTE_ORDER#_LOW_HIGH, AryOut:=iVarBin[0]);
				Inc(iVarIndex);
			195:
				iVarName := 'DT_ARR_D3_E1_LH';
				iVarDeclare := 'ARRAY[0..0,0..0,0..0] OF DATE_AND_TIME';
				// iVarValue := '[[["1970-01-01T00:00:00.0000001Z"]]]';
				iVarValue := '[[[100]]]';
				iVarKsType := 'nj::date_and_time_array_3d(1,1,1)';
				iVarKsId := 'date_and_time_arr_d3_e1_lh';
				
				Clear(DT_ARR_D3_E1);
				DT_ARR_D3_E1[0, 0, 0] := DT#1970-01-01-00:00:00.000000100;
				iVarBinSize := ToAryByte(In:=DT_ARR_D3_E1, Order:=_eBYTE_ORDER#_LOW_HIGH, AryOut:=iVarBin[0]);
				iVarIndex := iVarIndex - iVarIndex MOD 10 + 10;

			// Struct
			// Alignment1Struct
			200:
				iVarName := 'STRUCT_ALIGNMENT1';
				iVarDeclare := 'Alignment1Struct';
				iVarValue := '{"aSint":-1, "aUsint":2, "Bytes":[3,4]}';
				
				Clear(STRUCT_ALIGNMENT1);
				STRUCT_ALIGNMENT1.aSint := -1; STRUCT_ALIGNMENT1.aUsint := 2;
				STRUCT_ALIGNMENT1.Bytes[0] := 3; STRUCT_ALIGNMENT1.Bytes[1] := 4;
				iVarBinSize := ToAryByte(In:=STRUCT_ALIGNMENT1, Order:=_eBYTE_ORDER#_LOW_HIGH, AryOut:=iVarBin[0]);
				Inc(iVarIndex);
			201:
				iVarName := 'STRUCT_ALIGNMENT1_ARR_D1';
				iVarDeclare := 'ARRAY [0..2] OF Alignment1Struct';
				iVarValue := '[{"aSint":-1, "aUsint":2, "Bytes":[3,4]}, {"aSint":0, "aUsint":0, "Bytes":[0,0]}, {"aSint":-1, "aUsint":2, "Bytes":[3,4]}]';
				
				Clear(STRUCT_ALIGNMENT1_ARR_D1);
				STRUCT_ALIGNMENT1.aSint := -1; STRUCT_ALIGNMENT1.aUsint := 2;
				STRUCT_ALIGNMENT1.Bytes[0] := 3; STRUCT_ALIGNMENT1.Bytes[1] := 4;
				STRUCT_ALIGNMENT1_ARR_D1[0] := STRUCT_ALIGNMENT1; STRUCT_ALIGNMENT1_ARR_D1[2] := STRUCT_ALIGNMENT1;
				iVarBinSize := ToAryByte(In:=STRUCT_ALIGNMENT1_ARR_D1, Order:=_eBYTE_ORDER#_LOW_HIGH, AryOut:=iVarBin[0]);
				iVarIndex := iVarIndex - iVarIndex MOD 10 + 10;

			// Alignment2Struct
			210:
				iVarName := 'STRUCT_ALIGNMENT2';
				iVarDeclare := 'Alignment2Struct';
				iVarValue := '{"aBool":true, "aInt":-1, "aUint":2, "Bools":[true,false,false,true]}';
				
